// TIA Portal V16 export
// export: Created 2023-05-31T09:36:56.6738296Z, ExportSetting WithDefaults, DisplayName Totally Integrated Automation Portal, DisplayVersion V16 Update 3, DisplayName TIA Portal Version Control Interface, DisplayVersion V16 Update 2, DisplayName TIA Portal Openness, DisplayVersion V16 Update 3, DisplayName SINAMICS Startdrive Advanced, DisplayVersion V16, DisplayName SINAMICS Startdrive G130, G150, S120, S150, SINAMICS MV, S210, DisplayVersion V16, DisplayName SINAMICS Startdrive G110M, G120, G120C, G120D, G120P, DisplayVersion V16, DisplayName STEP 7 Professional, DisplayVersion V16 Update 3, DisplayName STEP 7 Safety, DisplayVersion V16, DisplayName WinCC Advanced, DisplayVersion V16 Update 3
FUNCTION "CIP LINEA 2" : Void   // FC54, LAD
{ S7_Optimized_Access := 'FALSE' }
VERSION : 0.1
// trabajo paralelo desde kjsdfgvjosod
// stored: AutoNumber false, IsIECCheckEnabled false, SetENOAutomatically false, UDAEnableTagReadback false
   VAR_TEMP   // added for the SCL form of the ladder/FBD networks
      _w1 : Bool;
      _s5time1 : S5Time;
   END_VAR
BEGIN

REGION Network 1: SOLO EN LIMPIEZA TANQUES
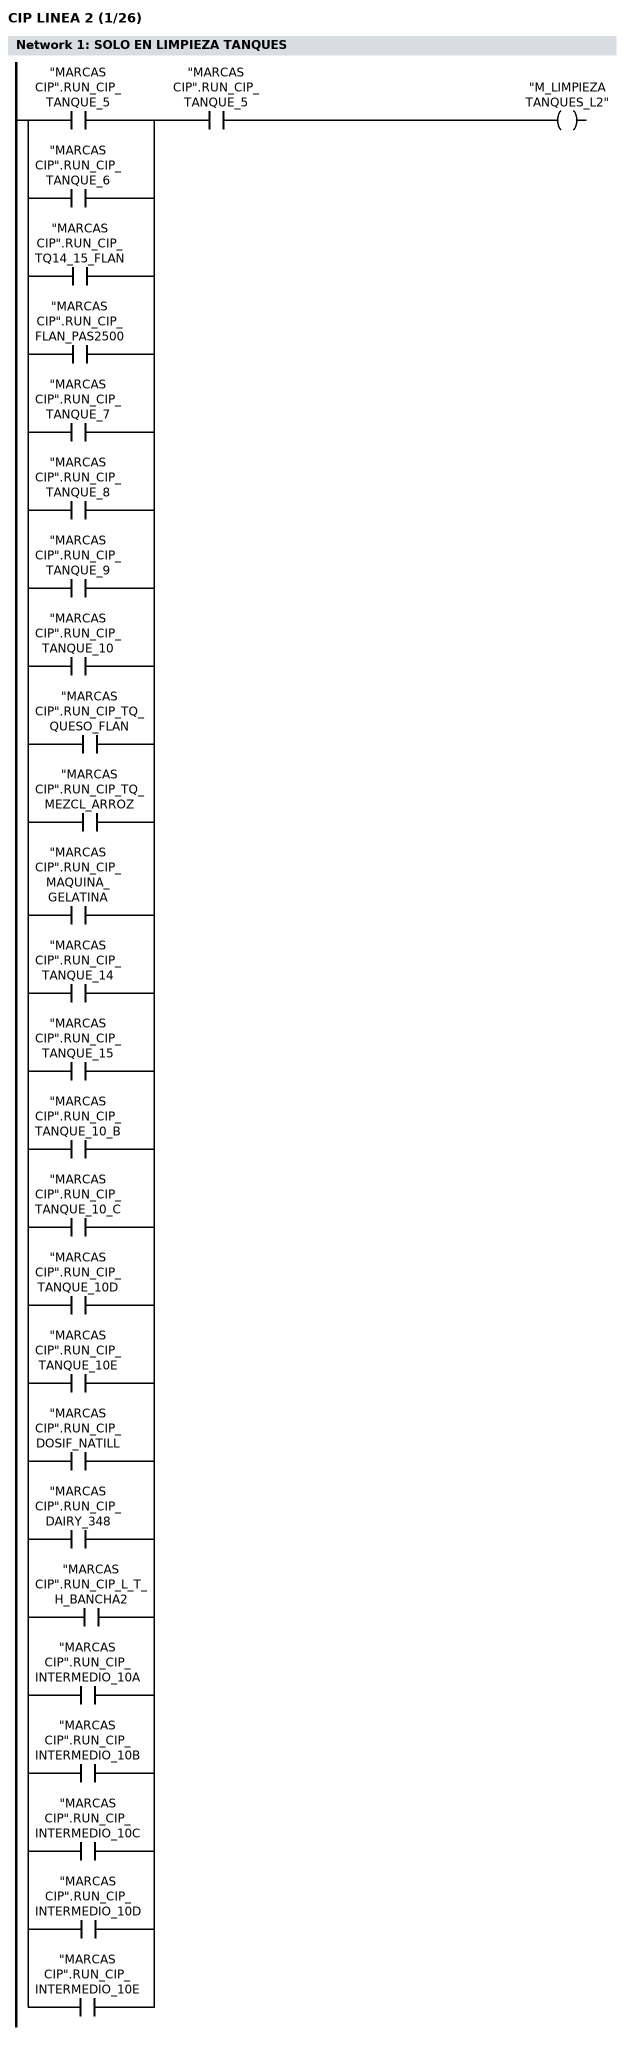
   RUNG wire#powerrail
      Contact( "MARCAS CIP".RUN_CIP_TANQUE_5 )
      wire#w1
      Contact( "MARCAS CIP".RUN_CIP_TANQUE_5 )
      Coil( "M_LIMPIEZA TANQUES_L2" )
   END_RUNG
   RUNG wire#powerrail
      Contact( "MARCAS CIP".RUN_CIP_TANQUE_6 )
   END_RUNG wire#w1
   RUNG wire#powerrail
      Contact( "MARCAS CIP".RUN_CIP_TQ14_15_FLAN )
   END_RUNG wire#w1
   RUNG wire#powerrail
      Contact( "MARCAS CIP".RUN_CIP_FLAN_PAS2500 )
   END_RUNG wire#w1
   RUNG wire#powerrail
      Contact( "MARCAS CIP".RUN_CIP_TANQUE_7 )
   END_RUNG wire#w1
   RUNG wire#powerrail
      Contact( "MARCAS CIP".RUN_CIP_TANQUE_8 )
   END_RUNG wire#w1
   RUNG wire#powerrail
      Contact( "MARCAS CIP".RUN_CIP_TANQUE_9 )
   END_RUNG wire#w1
   RUNG wire#powerrail
      Contact( "MARCAS CIP".RUN_CIP_TANQUE_10 )
   END_RUNG wire#w1
   RUNG wire#powerrail
      Contact( "MARCAS CIP".RUN_CIP_TQ_QUESO_FLAN )
   END_RUNG wire#w1
   RUNG wire#powerrail
      Contact( "MARCAS CIP".RUN_CIP_TQ_MEZCL_ARROZ )
   END_RUNG wire#w1
   RUNG wire#powerrail
      Contact( "MARCAS CIP".RUN_CIP_MAQUINA_GELATINA )
   END_RUNG wire#w1
   RUNG wire#powerrail
      Contact( "MARCAS CIP".RUN_CIP_TANQUE_14 )
   END_RUNG wire#w1
   RUNG wire#powerrail
      Contact( "MARCAS CIP".RUN_CIP_TANQUE_15 )
   END_RUNG wire#w1
   RUNG wire#powerrail
      Contact( "MARCAS CIP".RUN_CIP_TANQUE_10_B )
   END_RUNG wire#w1
   RUNG wire#powerrail
      Contact( "MARCAS CIP".RUN_CIP_TANQUE_10_C )
   END_RUNG wire#w1
   RUNG wire#powerrail
      Contact( "MARCAS CIP".RUN_CIP_TANQUE_10D )
   END_RUNG wire#w1
   RUNG wire#powerrail
      Contact( "MARCAS CIP".RUN_CIP_TANQUE_10E )
   END_RUNG wire#w1
   RUNG wire#powerrail
      Contact( "MARCAS CIP".RUN_CIP_DOSIF_NATILL )
   END_RUNG wire#w1
   RUNG wire#powerrail
      Contact( "MARCAS CIP".RUN_CIP_DAIRY_348 )
   END_RUNG wire#w1
   RUNG wire#powerrail
      Contact( "MARCAS CIP".RUN_CIP_L_T_H_BANCHA2 )
   END_RUNG wire#w1
   RUNG wire#powerrail
      Contact( "MARCAS CIP".RUN_CIP_INTERMEDIO_10A )
   END_RUNG wire#w1
   RUNG wire#powerrail
      Contact( "MARCAS CIP".RUN_CIP_INTERMEDIO_10B )
   END_RUNG wire#w1
   RUNG wire#powerrail
      Contact( "MARCAS CIP".RUN_CIP_INTERMEDIO_10C )
   END_RUNG wire#w1
   RUNG wire#powerrail
      Contact( "MARCAS CIP".RUN_CIP_INTERMEDIO_10D )
   END_RUNG wire#w1
   RUNG wire#powerrail
      Contact( "MARCAS CIP".RUN_CIP_INTERMEDIO_10E )
   END_RUNG wire#w1
   // the same network as SCL:
   "M_LIMPIEZA TANQUES_L2" := ("MARCAS CIP".RUN_CIP_TANQUE_5 OR "MARCAS CIP".RUN_CIP_TANQUE_6 OR "MARCAS CIP".RUN_CIP_TQ14_15_FLAN OR "MARCAS CIP".RUN_CIP_FLAN_PAS2500 OR "MARCAS CIP".RUN_CIP_TANQUE_7 OR "MARCAS CIP".RUN_CIP_TANQUE_8 OR "MARCAS CIP".RUN_CIP_TANQUE_9 OR "MARCAS CIP".RUN_CIP_TANQUE_10 OR "MARCAS CIP".RUN_CIP_TQ_QUESO_FLAN OR "MARCAS CIP".RUN_CIP_TQ_MEZCL_ARROZ OR "MARCAS CIP".RUN_CIP_MAQUINA_GELATINA OR "MARCAS CIP".RUN_CIP_TANQUE_14 OR "MARCAS CIP".RUN_CIP_TANQUE_15 OR "MARCAS CIP".RUN_CIP_TANQUE_10_B OR "MARCAS CIP".RUN_CIP_TANQUE_10_C OR "MARCAS CIP".RUN_CIP_TANQUE_10D OR "MARCAS CIP".RUN_CIP_TANQUE_10E OR "MARCAS CIP".RUN_CIP_DOSIF_NATILL OR "MARCAS CIP".RUN_CIP_DAIRY_348 OR "MARCAS CIP".RUN_CIP_L_T_H_BANCHA2 OR "MARCAS CIP".RUN_CIP_INTERMEDIO_10A OR "MARCAS CIP".RUN_CIP_INTERMEDIO_10B OR "MARCAS CIP".RUN_CIP_INTERMEDIO_10C OR "MARCAS CIP".RUN_CIP_INTERMEDIO_10D OR "MARCAS CIP".RUN_CIP_INTERMEDIO_10E) AND "MARCAS CIP".RUN_CIP_TANQUE_5;
END_REGION

REGION Network 2: PASO 1 PRIEMER ENJUAGUE AGUA RECUPERADA
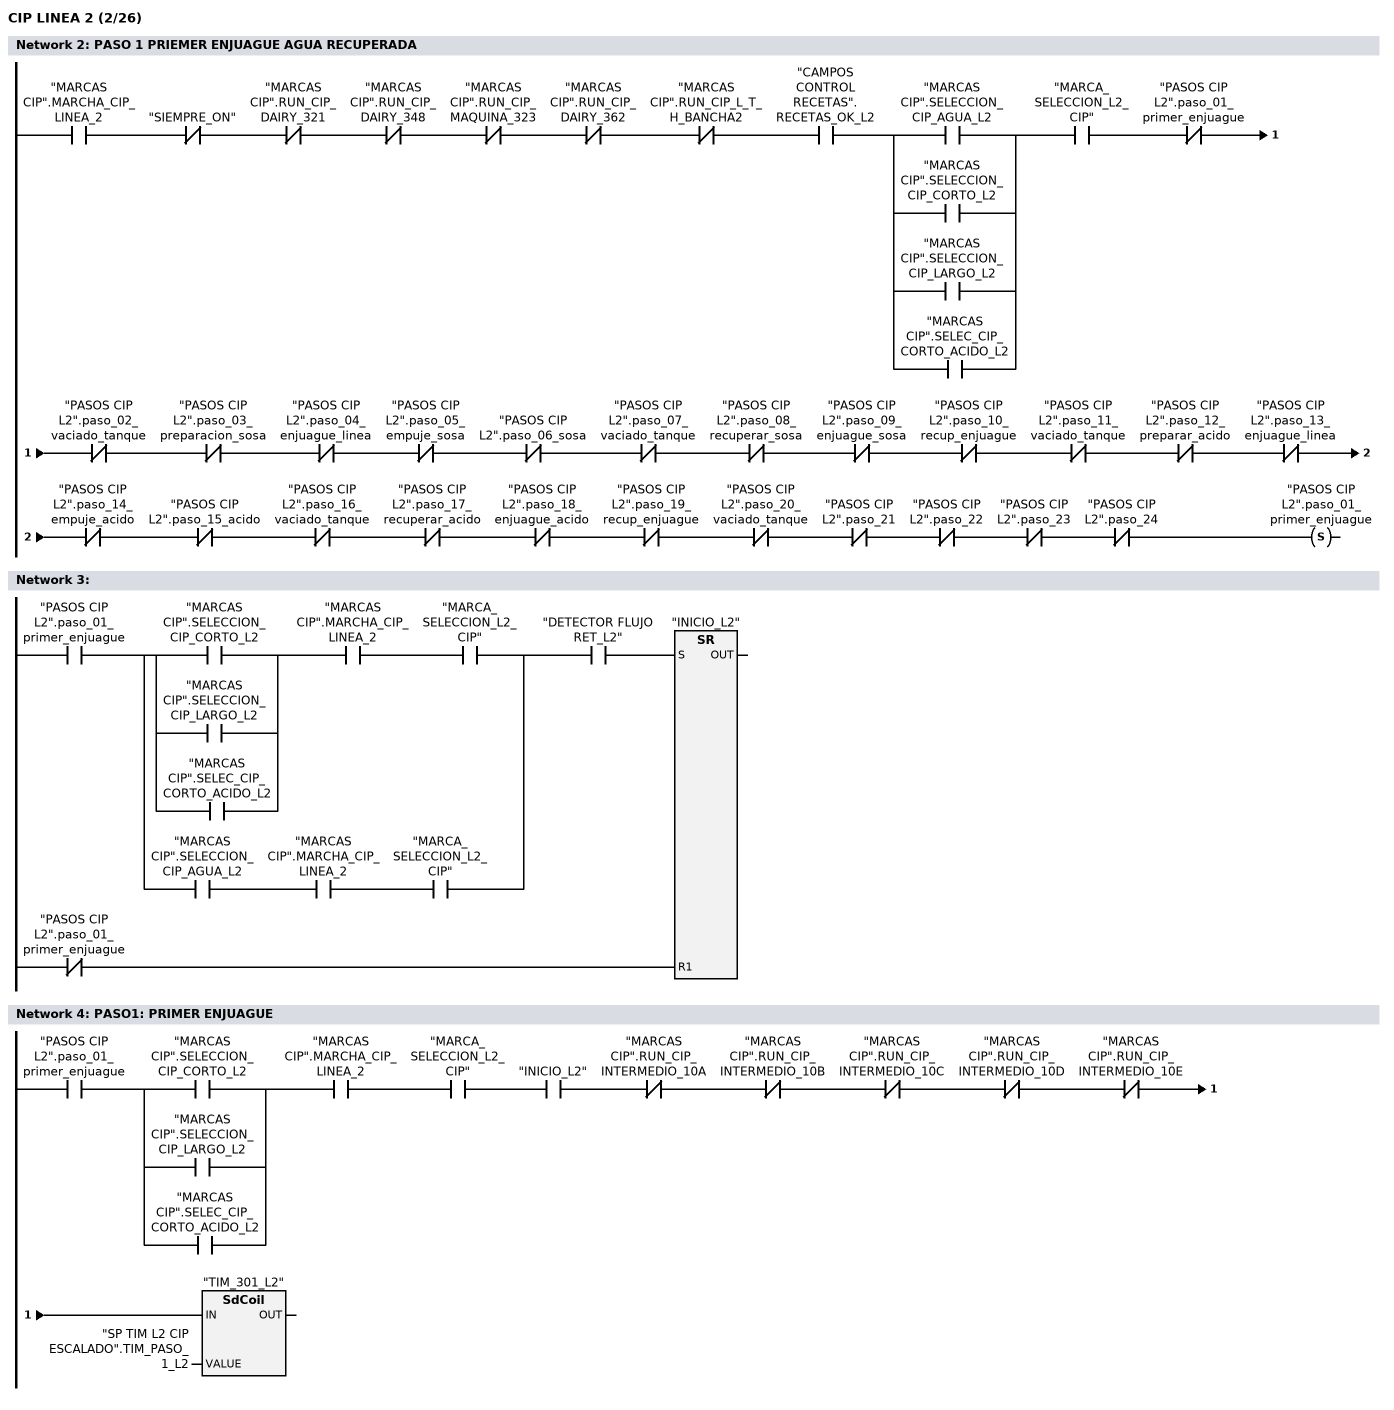
   RUNG wire#powerrail
      Contact( "MARCAS CIP".MARCHA_CIP_LINEA_2 )
      I_Contact( "SIEMPRE_ON" )
      I_Contact( "MARCAS CIP".RUN_CIP_DAIRY_321 )
      I_Contact( "MARCAS CIP".RUN_CIP_DAIRY_348 )
      I_Contact( "MARCAS CIP".RUN_CIP_MAQUINA_323 )
      I_Contact( "MARCAS CIP".RUN_CIP_DAIRY_362 )
      I_Contact( "MARCAS CIP".RUN_CIP_L_T_H_BANCHA2 )
      Contact( "CAMPOS CONTROL RECETAS".RECETAS_OK_L2 )
      wire#w1
      Contact( "MARCAS CIP".SELECCION_CIP_AGUA_L2 )
      wire#w2
      Contact( "MARCA_SELECCION_L2_CIP" )
      I_Contact( "PASOS CIP L2".paso_01_primer_enjuague )
      I_Contact( "PASOS CIP L2".paso_02_vaciado_tanque )
      I_Contact( "PASOS CIP L2".paso_03_preparacion_sosa )
      I_Contact( "PASOS CIP L2".paso_04_enjuague_linea )
      I_Contact( "PASOS CIP L2".paso_05_empuje_sosa )
      I_Contact( "PASOS CIP L2".paso_06_sosa )
      I_Contact( "PASOS CIP L2".paso_07_vaciado_tanque )
      I_Contact( "PASOS CIP L2".paso_08_recuperar_sosa )
      I_Contact( "PASOS CIP L2".paso_09_enjuague_sosa )
      I_Contact( "PASOS CIP L2".paso_10_recup_enjuague )
      I_Contact( "PASOS CIP L2".paso_11_vaciado_tanque )
      I_Contact( "PASOS CIP L2".paso_12_preparar_acido )
      I_Contact( "PASOS CIP L2".paso_13_enjuague_linea )
      I_Contact( "PASOS CIP L2".paso_14_empuje_acido )
      I_Contact( "PASOS CIP L2".paso_15_acido )
      I_Contact( "PASOS CIP L2".paso_16_vaciado_tanque )
      I_Contact( "PASOS CIP L2".paso_17_recuperar_acido )
      I_Contact( "PASOS CIP L2".paso_18_enjuague_acido )
      I_Contact( "PASOS CIP L2".paso_19_recup_enjuague )
      I_Contact( "PASOS CIP L2".paso_20_vaciado_tanque )
      I_Contact( "PASOS CIP L2".paso_21 )
      I_Contact( "PASOS CIP L2".paso_22 )
      I_Contact( "PASOS CIP L2".paso_23 )
      I_Contact( "PASOS CIP L2".paso_24 )
      S_Coil( "PASOS CIP L2".paso_01_primer_enjuague )
   END_RUNG
   RUNG wire#w1
      Contact( "MARCAS CIP".SELECCION_CIP_CORTO_L2 )
   END_RUNG wire#w2
   RUNG wire#w1
      Contact( "MARCAS CIP".SELECCION_CIP_LARGO_L2 )
   END_RUNG wire#w2
   RUNG wire#w1
      Contact( "MARCAS CIP".SELEC_CIP_CORTO_ACIDO_L2 )
   END_RUNG wire#w2
   // the same network as SCL:
   IF "MARCAS CIP".MARCHA_CIP_LINEA_2 AND NOT "SIEMPRE_ON" AND NOT "MARCAS CIP".RUN_CIP_DAIRY_321 AND NOT "MARCAS CIP".RUN_CIP_DAIRY_348 AND NOT "MARCAS CIP".RUN_CIP_MAQUINA_323 AND NOT "MARCAS CIP".RUN_CIP_DAIRY_362 AND NOT "MARCAS CIP".RUN_CIP_L_T_H_BANCHA2 AND "CAMPOS CONTROL RECETAS".RECETAS_OK_L2 AND ("MARCAS CIP".SELECCION_CIP_AGUA_L2 OR "MARCAS CIP".SELECCION_CIP_CORTO_L2 OR "MARCAS CIP".SELECCION_CIP_LARGO_L2 OR "MARCAS CIP".SELEC_CIP_CORTO_ACIDO_L2) AND "MARCA_SELECCION_L2_CIP" AND NOT "PASOS CIP L2".paso_01_primer_enjuague AND NOT "PASOS CIP L2".paso_02_vaciado_tanque AND NOT "PASOS CIP L2".paso_03_preparacion_sosa AND NOT "PASOS CIP L2".paso_04_enjuague_linea AND NOT "PASOS CIP L2".paso_05_empuje_sosa AND NOT "PASOS CIP L2".paso_06_sosa AND NOT "PASOS CIP L2".paso_07_vaciado_tanque AND NOT "PASOS CIP L2".paso_08_recuperar_sosa AND NOT "PASOS CIP L2".paso_09_enjuague_sosa AND NOT "PASOS CIP L2".paso_10_recup_enjuague AND NOT "PASOS CIP L2".paso_11_vaciado_tanque AND NOT "PASOS CIP L2".paso_12_preparar_acido AND NOT "PASOS CIP L2".paso_13_enjuague_linea AND NOT "PASOS CIP L2".paso_14_empuje_acido AND NOT "PASOS CIP L2".paso_15_acido AND NOT "PASOS CIP L2".paso_16_vaciado_tanque AND NOT "PASOS CIP L2".paso_17_recuperar_acido AND NOT "PASOS CIP L2".paso_18_enjuague_acido AND NOT "PASOS CIP L2".paso_19_recup_enjuague AND NOT "PASOS CIP L2".paso_20_vaciado_tanque AND NOT "PASOS CIP L2".paso_21 AND NOT "PASOS CIP L2".paso_22 AND NOT "PASOS CIP L2".paso_23 AND NOT "PASOS CIP L2".paso_24 THEN
       "PASOS CIP L2".paso_01_primer_enjuague := TRUE;
   END_IF;
END_REGION

REGION Network 3
   RUNG wire#powerrail
      Contact( "PASOS CIP L2".paso_01_primer_enjuague )
      wire#w1
      Contact( "MARCAS CIP".SELECCION_CIP_CORTO_L2 )
      wire#w2
      Contact( "MARCAS CIP".MARCHA_CIP_LINEA_2 )
      Contact( "MARCA_SELECCION_L2_CIP" )
      wire#w3
      Contact( "DETECTOR FLUJO RET_L2" )
      S_SR(operand := "INICIO_L2", r1 := wire#w4)
   END_RUNG
   RUNG wire#w1
      Contact( "MARCAS CIP".SELECCION_CIP_LARGO_L2 )
   END_RUNG wire#w2
   RUNG wire#w1
      Contact( "MARCAS CIP".SELEC_CIP_CORTO_ACIDO_L2 )
   END_RUNG wire#w2
   RUNG wire#w1
      Contact( "MARCAS CIP".SELECCION_CIP_AGUA_L2 )
      Contact( "MARCAS CIP".MARCHA_CIP_LINEA_2 )
      Contact( "MARCA_SELECCION_L2_CIP" )
   END_RUNG wire#w3
   RUNG wire#powerrail
      I_Contact( "PASOS CIP L2".paso_01_primer_enjuague )
   END_RUNG wire#w4
   // the same network as SCL:
   IF "PASOS CIP L2".paso_01_primer_enjuague AND ((("MARCAS CIP".SELECCION_CIP_CORTO_L2 OR "MARCAS CIP".SELECCION_CIP_LARGO_L2 OR "MARCAS CIP".SELEC_CIP_CORTO_ACIDO_L2) AND "MARCAS CIP".MARCHA_CIP_LINEA_2 AND "MARCA_SELECCION_L2_CIP") OR ("MARCAS CIP".SELECCION_CIP_AGUA_L2 AND "MARCAS CIP".MARCHA_CIP_LINEA_2 AND "MARCA_SELECCION_L2_CIP")) AND "DETECTOR FLUJO RET_L2" THEN
       "INICIO_L2" := TRUE;   // SR flip-flop
   END_IF;
   IF NOT "PASOS CIP L2".paso_01_primer_enjuague THEN "INICIO_L2" := FALSE; END_IF;
END_REGION

REGION Network 4: PASO1: PRIMER ENJUAGUE
   // no SCL statement known for SdCoil: written as a call
   SdCoil(value := "SP TIM L2 CIP ESCALADO".TIM_PASO_1_L2,
          operand := "TIM_301_L2",
          in := "PASOS CIP L2".paso_01_primer_enjuague AND ("MARCAS CIP".SELECCION_CIP_CORTO_L2 OR "MARCAS CIP".SELECCION_CIP_LARGO_L2 OR "MARCAS CIP".SELEC_CIP_CORTO_ACIDO_L2) AND "MARCAS CIP".MARCHA_CIP_LINEA_2 AND "MARCA_SELECCION_L2_CIP" AND "INICIO_L2" AND NOT "MARCAS CIP".RUN_CIP_INTERMEDIO_10A AND NOT "MARCAS CIP".RUN_CIP_INTERMEDIO_10B AND NOT "MARCAS CIP".RUN_CIP_INTERMEDIO_10C AND NOT "MARCAS CIP".RUN_CIP_INTERMEDIO_10D AND NOT "MARCAS CIP".RUN_CIP_INTERMEDIO_10E);
END_REGION

REGION Network 5: PASO 2: VACIADO TANQUE (SOLO BOMBA RETORNO CIP)
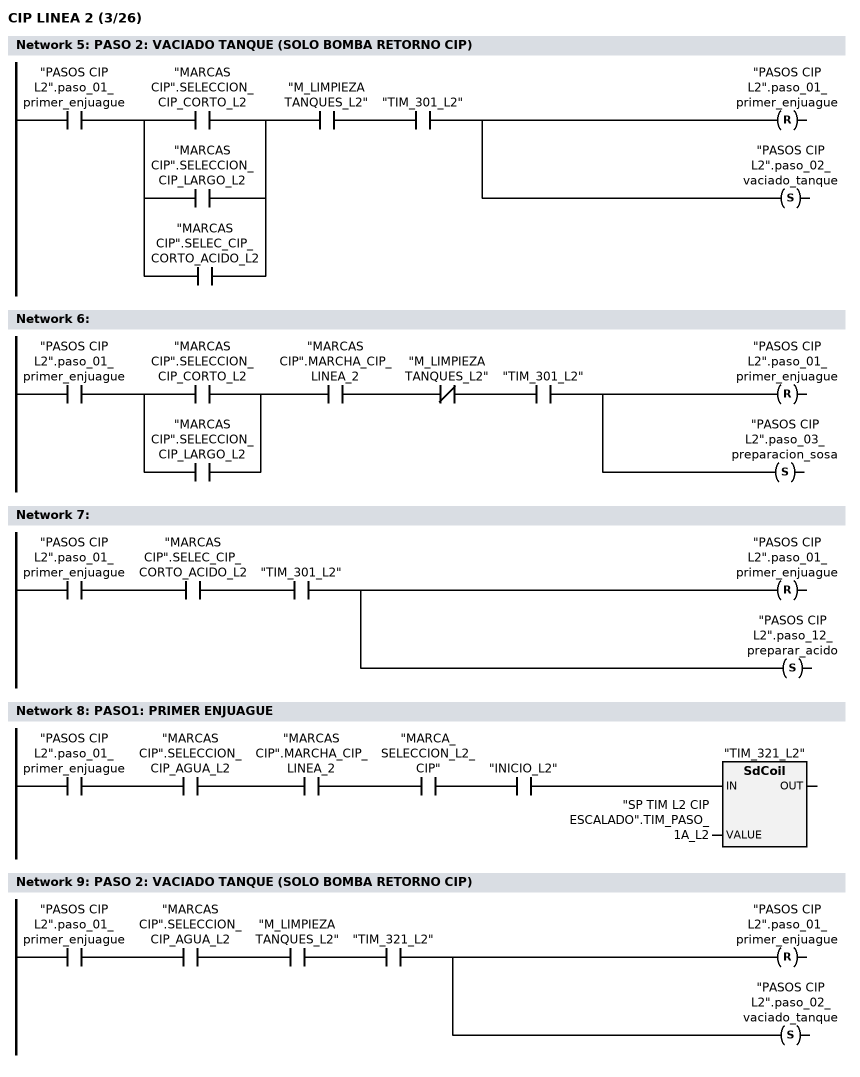
   RUNG wire#powerrail
      Contact( "PASOS CIP L2".paso_01_primer_enjuague )
      wire#w1
      Contact( "MARCAS CIP".SELECCION_CIP_CORTO_L2 )
      wire#w2
      Contact( "M_LIMPIEZA TANQUES_L2" )
      Contact( "TIM_301_L2" )
      wire#w3
      R_Coil( "PASOS CIP L2".paso_01_primer_enjuague )
   END_RUNG
   RUNG wire#w1
      Contact( "MARCAS CIP".SELECCION_CIP_LARGO_L2 )
   END_RUNG wire#w2
   RUNG wire#w1
      Contact( "MARCAS CIP".SELEC_CIP_CORTO_ACIDO_L2 )
   END_RUNG wire#w2
   RUNG wire#w3
      S_Coil( "PASOS CIP L2".paso_02_vaciado_tanque )
   END_RUNG
   // the same network as SCL:
   #_w1 := "PASOS CIP L2".paso_01_primer_enjuague AND ("MARCAS CIP".SELECCION_CIP_CORTO_L2 OR "MARCAS CIP".SELECCION_CIP_LARGO_L2 OR "MARCAS CIP".SELEC_CIP_CORTO_ACIDO_L2) AND "M_LIMPIEZA TANQUES_L2" AND "TIM_301_L2";
   IF #_w1 THEN
       "PASOS CIP L2".paso_01_primer_enjuague := FALSE;
       "PASOS CIP L2".paso_02_vaciado_tanque := TRUE;
   END_IF;
END_REGION

REGION Network 6
   RUNG wire#powerrail
      Contact( "PASOS CIP L2".paso_01_primer_enjuague )
      wire#w1
      Contact( "MARCAS CIP".SELECCION_CIP_CORTO_L2 )
      wire#w2
      Contact( "MARCAS CIP".MARCHA_CIP_LINEA_2 )
      I_Contact( "M_LIMPIEZA TANQUES_L2" )
      Contact( "TIM_301_L2" )
      wire#w3
      R_Coil( "PASOS CIP L2".paso_01_primer_enjuague )
   END_RUNG
   RUNG wire#w1
      Contact( "MARCAS CIP".SELECCION_CIP_LARGO_L2 )
   END_RUNG wire#w2
   RUNG wire#w3
      S_Coil( "PASOS CIP L2".paso_03_preparacion_sosa )
   END_RUNG
   // the same network as SCL:
   #_w1 := "PASOS CIP L2".paso_01_primer_enjuague AND ("MARCAS CIP".SELECCION_CIP_CORTO_L2 OR "MARCAS CIP".SELECCION_CIP_LARGO_L2) AND "MARCAS CIP".MARCHA_CIP_LINEA_2 AND NOT "M_LIMPIEZA TANQUES_L2" AND "TIM_301_L2";
   IF #_w1 THEN
       "PASOS CIP L2".paso_01_primer_enjuague := FALSE;
       "PASOS CIP L2".paso_03_preparacion_sosa := TRUE;
   END_IF;
END_REGION

REGION Network 7
   RUNG wire#powerrail
      Contact( "PASOS CIP L2".paso_01_primer_enjuague )
      Contact( "MARCAS CIP".SELEC_CIP_CORTO_ACIDO_L2 )
      Contact( "TIM_301_L2" )
      wire#w1
      R_Coil( "PASOS CIP L2".paso_01_primer_enjuague )
   END_RUNG
   RUNG wire#w1
      S_Coil( "PASOS CIP L2".paso_12_preparar_acido )
   END_RUNG
   // the same network as SCL:
   #_w1 := "PASOS CIP L2".paso_01_primer_enjuague AND "MARCAS CIP".SELEC_CIP_CORTO_ACIDO_L2 AND "TIM_301_L2";
   IF #_w1 THEN
       "PASOS CIP L2".paso_01_primer_enjuague := FALSE;
       "PASOS CIP L2".paso_12_preparar_acido := TRUE;
   END_IF;
END_REGION

REGION Network 8: PASO1: PRIMER ENJUAGUE
   // no SCL statement known for SdCoil: written as a call
   SdCoil(value := "SP TIM L2 CIP ESCALADO".TIM_PASO_1A_L2,
          operand := "TIM_321_L2",
          in := "PASOS CIP L2".paso_01_primer_enjuague AND "MARCAS CIP".SELECCION_CIP_AGUA_L2 AND "MARCAS CIP".MARCHA_CIP_LINEA_2 AND "MARCA_SELECCION_L2_CIP" AND "INICIO_L2");
END_REGION

REGION Network 9: PASO 2: VACIADO TANQUE (SOLO BOMBA RETORNO CIP)
   RUNG wire#powerrail
      Contact( "PASOS CIP L2".paso_01_primer_enjuague )
      Contact( "MARCAS CIP".SELECCION_CIP_AGUA_L2 )
      Contact( "M_LIMPIEZA TANQUES_L2" )
      Contact( "TIM_321_L2" )
      wire#w1
      R_Coil( "PASOS CIP L2".paso_01_primer_enjuague )
   END_RUNG
   RUNG wire#w1
      S_Coil( "PASOS CIP L2".paso_02_vaciado_tanque )
   END_RUNG
   // the same network as SCL:
   #_w1 := "PASOS CIP L2".paso_01_primer_enjuague AND "MARCAS CIP".SELECCION_CIP_AGUA_L2 AND "M_LIMPIEZA TANQUES_L2" AND "TIM_321_L2";
   IF #_w1 THEN
       "PASOS CIP L2".paso_01_primer_enjuague := FALSE;
       "PASOS CIP L2".paso_02_vaciado_tanque := TRUE;
   END_IF;
END_REGION

REGION Network 10
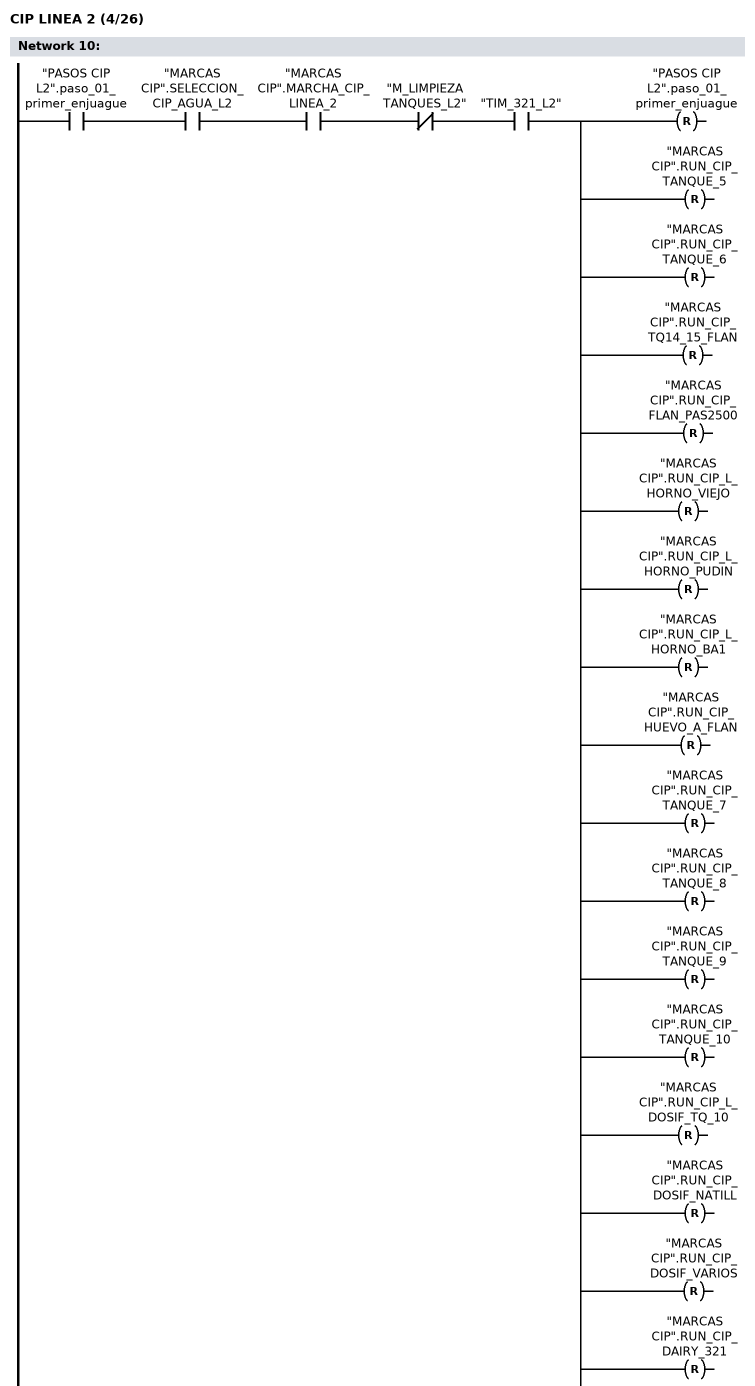
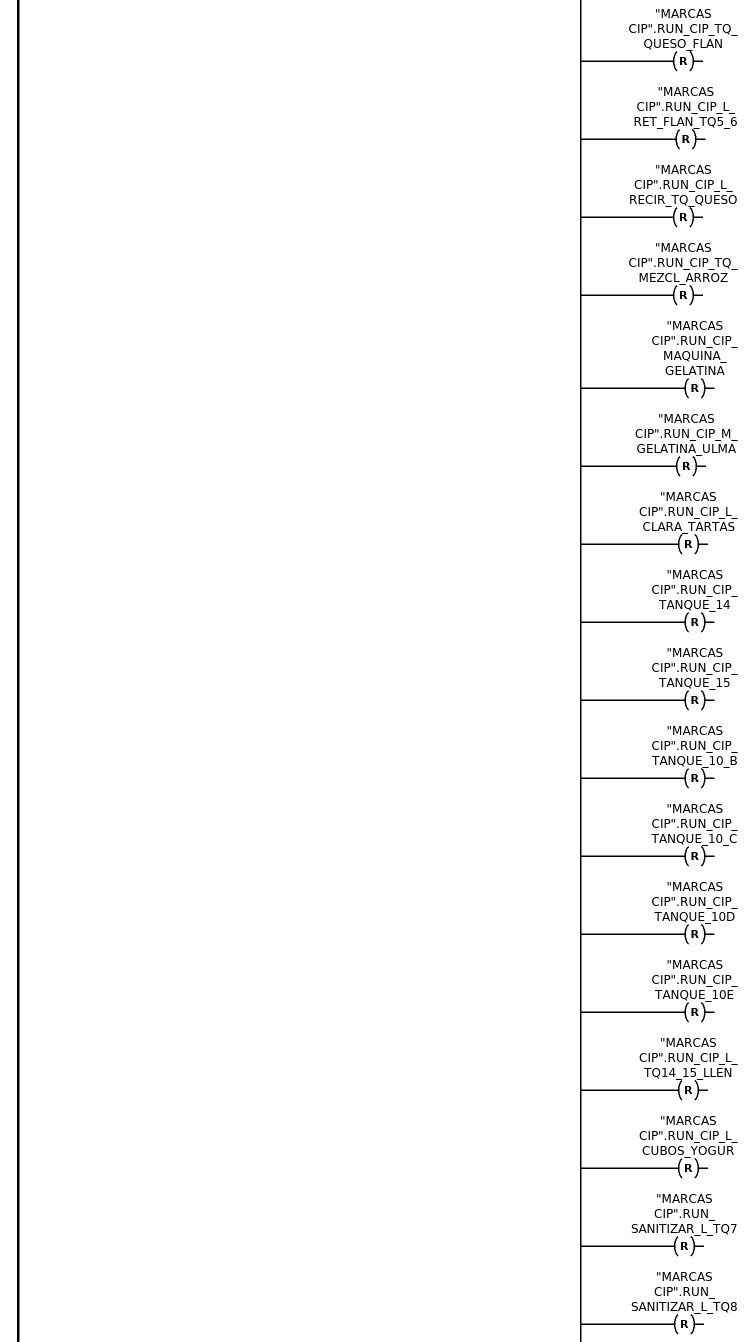
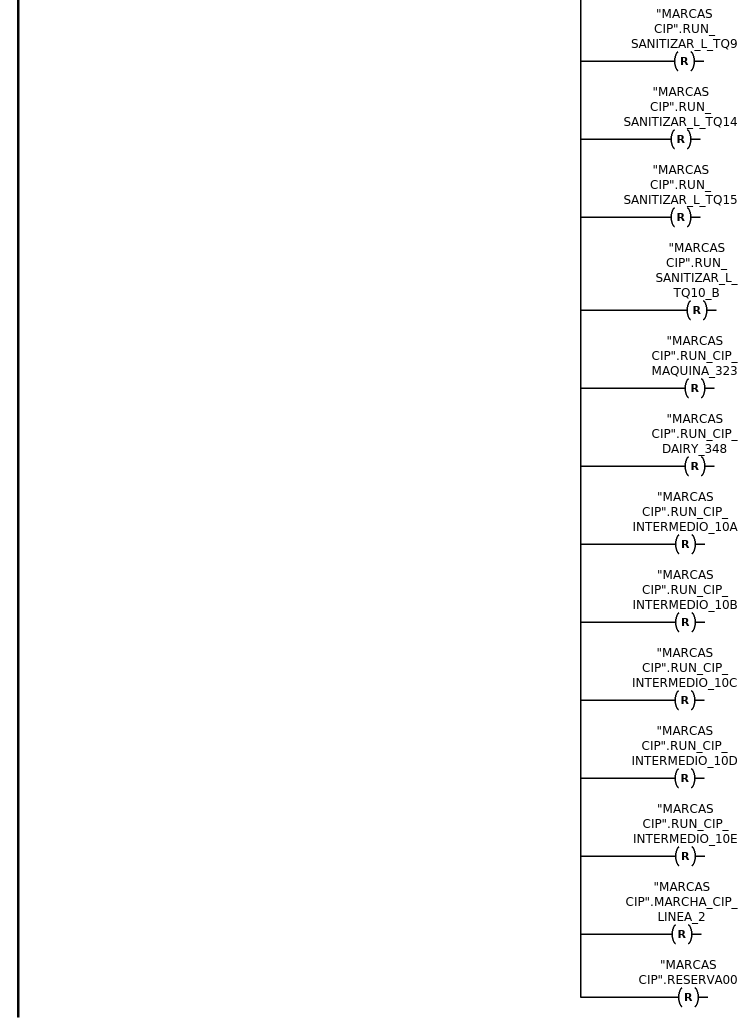
   RUNG wire#powerrail
      Contact( "PASOS CIP L2".paso_01_primer_enjuague )
      Contact( "MARCAS CIP".SELECCION_CIP_AGUA_L2 )
      Contact( "MARCAS CIP".MARCHA_CIP_LINEA_2 )
      I_Contact( "M_LIMPIEZA TANQUES_L2" )
      Contact( "TIM_321_L2" )
      wire#w1
      R_Coil( "PASOS CIP L2".paso_01_primer_enjuague )
   END_RUNG
   RUNG wire#w1
      R_Coil( "MARCAS CIP".RUN_CIP_TANQUE_5 )
   END_RUNG
   RUNG wire#w1
      R_Coil( "MARCAS CIP".RUN_CIP_TANQUE_6 )
   END_RUNG
   RUNG wire#w1
      R_Coil( "MARCAS CIP".RUN_CIP_TQ14_15_FLAN )
   END_RUNG
   RUNG wire#w1
      R_Coil( "MARCAS CIP".RUN_CIP_FLAN_PAS2500 )
   END_RUNG
   RUNG wire#w1
      R_Coil( "MARCAS CIP".RUN_CIP_L_HORNO_VIEJO )
   END_RUNG
   RUNG wire#w1
      R_Coil( "MARCAS CIP".RUN_CIP_L_HORNO_PUDIN )
   END_RUNG
   RUNG wire#w1
      R_Coil( "MARCAS CIP".RUN_CIP_L_HORNO_BA1 )
   END_RUNG
   RUNG wire#w1
      R_Coil( "MARCAS CIP".RUN_CIP_HUEVO_A_FLAN )
   END_RUNG
   RUNG wire#w1
      R_Coil( "MARCAS CIP".RUN_CIP_TANQUE_7 )
   END_RUNG
   RUNG wire#w1
      R_Coil( "MARCAS CIP".RUN_CIP_TANQUE_8 )
   END_RUNG
   RUNG wire#w1
      R_Coil( "MARCAS CIP".RUN_CIP_TANQUE_9 )
   END_RUNG
   RUNG wire#w1
      R_Coil( "MARCAS CIP".RUN_CIP_TANQUE_10 )
   END_RUNG
   RUNG wire#w1
      R_Coil( "MARCAS CIP".RUN_CIP_L_DOSIF_TQ_10 )
   END_RUNG
   RUNG wire#w1
      R_Coil( "MARCAS CIP".RUN_CIP_DOSIF_NATILL )
   END_RUNG
   RUNG wire#w1
      R_Coil( "MARCAS CIP".RUN_CIP_DOSIF_VARIOS )
   END_RUNG
   RUNG wire#w1
      R_Coil( "MARCAS CIP".RUN_CIP_DAIRY_321 )
   END_RUNG
   RUNG wire#w1
      R_Coil( "MARCAS CIP".RUN_CIP_TQ_QUESO_FLAN )
   END_RUNG
   RUNG wire#w1
      R_Coil( "MARCAS CIP".RUN_CIP_L_RET_FLAN_TQ5_6 )
   END_RUNG
   RUNG wire#w1
      R_Coil( "MARCAS CIP".RUN_CIP_L_RECIR_TQ_QUESO )
   END_RUNG
   RUNG wire#w1
      R_Coil( "MARCAS CIP".RUN_CIP_TQ_MEZCL_ARROZ )
   END_RUNG
   RUNG wire#w1
      R_Coil( "MARCAS CIP".RUN_CIP_MAQUINA_GELATINA )
   END_RUNG
   RUNG wire#w1
      R_Coil( "MARCAS CIP".RUN_CIP_M_GELATINA_ULMA )
   END_RUNG
   RUNG wire#w1
      R_Coil( "MARCAS CIP".RUN_CIP_L_CLARA_TARTAS )
   END_RUNG
   RUNG wire#w1
      R_Coil( "MARCAS CIP".RUN_CIP_TANQUE_14 )
   END_RUNG
   RUNG wire#w1
      R_Coil( "MARCAS CIP".RUN_CIP_TANQUE_15 )
   END_RUNG
   RUNG wire#w1
      R_Coil( "MARCAS CIP".RUN_CIP_TANQUE_10_B )
   END_RUNG
   RUNG wire#w1
      R_Coil( "MARCAS CIP".RUN_CIP_TANQUE_10_C )
   END_RUNG
   RUNG wire#w1
      R_Coil( "MARCAS CIP".RUN_CIP_TANQUE_10D )
   END_RUNG
   RUNG wire#w1
      R_Coil( "MARCAS CIP".RUN_CIP_TANQUE_10E )
   END_RUNG
   RUNG wire#w1
      R_Coil( "MARCAS CIP".RUN_CIP_L_TQ14_15_LLEN )
   END_RUNG
   RUNG wire#w1
      R_Coil( "MARCAS CIP".RUN_CIP_L_CUBOS_YOGUR )
   END_RUNG
   RUNG wire#w1
      R_Coil( "MARCAS CIP".RUN_SANITIZAR_L_TQ7 )
   END_RUNG
   RUNG wire#w1
      R_Coil( "MARCAS CIP".RUN_SANITIZAR_L_TQ8 )
   END_RUNG
   RUNG wire#w1
      R_Coil( "MARCAS CIP".RUN_SANITIZAR_L_TQ9 )
   END_RUNG
   RUNG wire#w1
      R_Coil( "MARCAS CIP".RUN_SANITIZAR_L_TQ14 )
   END_RUNG
   RUNG wire#w1
      R_Coil( "MARCAS CIP".RUN_SANITIZAR_L_TQ15 )
   END_RUNG
   RUNG wire#w1
      R_Coil( "MARCAS CIP".RUN_SANITIZAR_L_TQ10_B )
   END_RUNG
   RUNG wire#w1
      R_Coil( "MARCAS CIP".RUN_CIP_MAQUINA_323 )
   END_RUNG
   RUNG wire#w1
      R_Coil( "MARCAS CIP".RUN_CIP_DAIRY_348 )
   END_RUNG
   RUNG wire#w1
      R_Coil( "MARCAS CIP".RUN_CIP_INTERMEDIO_10A )
   END_RUNG
   RUNG wire#w1
      R_Coil( "MARCAS CIP".RUN_CIP_INTERMEDIO_10B )
   END_RUNG
   RUNG wire#w1
      R_Coil( "MARCAS CIP".RUN_CIP_INTERMEDIO_10C )
   END_RUNG
   RUNG wire#w1
      R_Coil( "MARCAS CIP".RUN_CIP_INTERMEDIO_10D )
   END_RUNG
   RUNG wire#w1
      R_Coil( "MARCAS CIP".RUN_CIP_INTERMEDIO_10E )
   END_RUNG
   RUNG wire#w1
      R_Coil( "MARCAS CIP".MARCHA_CIP_LINEA_2 )
   END_RUNG
   RUNG wire#w1
      R_Coil( "MARCAS CIP".RESERVA00 )
   END_RUNG
   // the same network as SCL:
   #_w1 := "PASOS CIP L2".paso_01_primer_enjuague AND "MARCAS CIP".SELECCION_CIP_AGUA_L2 AND "MARCAS CIP".MARCHA_CIP_LINEA_2 AND NOT "M_LIMPIEZA TANQUES_L2" AND "TIM_321_L2";
   IF #_w1 THEN
       "PASOS CIP L2".paso_01_primer_enjuague := FALSE;
       "MARCAS CIP".RUN_CIP_TANQUE_5 := FALSE;
       "MARCAS CIP".RUN_CIP_TANQUE_6 := FALSE;
       "MARCAS CIP".RUN_CIP_TQ14_15_FLAN := FALSE;
       "MARCAS CIP".RUN_CIP_FLAN_PAS2500 := FALSE;
       "MARCAS CIP".RUN_CIP_L_HORNO_VIEJO := FALSE;
       "MARCAS CIP".RUN_CIP_L_HORNO_PUDIN := FALSE;
       "MARCAS CIP".RUN_CIP_L_HORNO_BA1 := FALSE;
       "MARCAS CIP".RUN_CIP_HUEVO_A_FLAN := FALSE;
       "MARCAS CIP".RUN_CIP_TANQUE_7 := FALSE;
       "MARCAS CIP".RUN_CIP_TANQUE_8 := FALSE;
       "MARCAS CIP".RUN_CIP_TANQUE_9 := FALSE;
       "MARCAS CIP".RUN_CIP_TANQUE_10 := FALSE;
       "MARCAS CIP".RUN_CIP_L_DOSIF_TQ_10 := FALSE;
       "MARCAS CIP".RUN_CIP_DOSIF_NATILL := FALSE;
       "MARCAS CIP".RUN_CIP_DOSIF_VARIOS := FALSE;
       "MARCAS CIP".RUN_CIP_DAIRY_321 := FALSE;
       "MARCAS CIP".RUN_CIP_TQ_QUESO_FLAN := FALSE;
       "MARCAS CIP".RUN_CIP_L_RET_FLAN_TQ5_6 := FALSE;
       "MARCAS CIP".RUN_CIP_L_RECIR_TQ_QUESO := FALSE;
       "MARCAS CIP".RUN_CIP_TQ_MEZCL_ARROZ := FALSE;
       "MARCAS CIP".RUN_CIP_MAQUINA_GELATINA := FALSE;
       "MARCAS CIP".RUN_CIP_M_GELATINA_ULMA := FALSE;
       "MARCAS CIP".RUN_CIP_L_CLARA_TARTAS := FALSE;
       "MARCAS CIP".RUN_CIP_TANQUE_14 := FALSE;
       "MARCAS CIP".RUN_CIP_TANQUE_15 := FALSE;
       "MARCAS CIP".RUN_CIP_TANQUE_10_B := FALSE;
       "MARCAS CIP".RUN_CIP_TANQUE_10_C := FALSE;
       "MARCAS CIP".RUN_CIP_TANQUE_10D := FALSE;
       "MARCAS CIP".RUN_CIP_TANQUE_10E := FALSE;
       "MARCAS CIP".RUN_CIP_L_TQ14_15_LLEN := FALSE;
       "MARCAS CIP".RUN_CIP_L_CUBOS_YOGUR := FALSE;
       "MARCAS CIP".RUN_SANITIZAR_L_TQ7 := FALSE;
       "MARCAS CIP".RUN_SANITIZAR_L_TQ8 := FALSE;
       "MARCAS CIP".RUN_SANITIZAR_L_TQ9 := FALSE;
       "MARCAS CIP".RUN_SANITIZAR_L_TQ14 := FALSE;
       "MARCAS CIP".RUN_SANITIZAR_L_TQ15 := FALSE;
       "MARCAS CIP".RUN_SANITIZAR_L_TQ10_B := FALSE;
       "MARCAS CIP".RUN_CIP_MAQUINA_323 := FALSE;
       "MARCAS CIP".RUN_CIP_DAIRY_348 := FALSE;
       "MARCAS CIP".RUN_CIP_INTERMEDIO_10A := FALSE;
       "MARCAS CIP".RUN_CIP_INTERMEDIO_10B := FALSE;
       "MARCAS CIP".RUN_CIP_INTERMEDIO_10C := FALSE;
       "MARCAS CIP".RUN_CIP_INTERMEDIO_10D := FALSE;
       "MARCAS CIP".RUN_CIP_INTERMEDIO_10E := FALSE;
       "MARCAS CIP".MARCHA_CIP_LINEA_2 := FALSE;
       "MARCAS CIP".RESERVA00 := FALSE;
   END_IF;
END_REGION

REGION Network 11
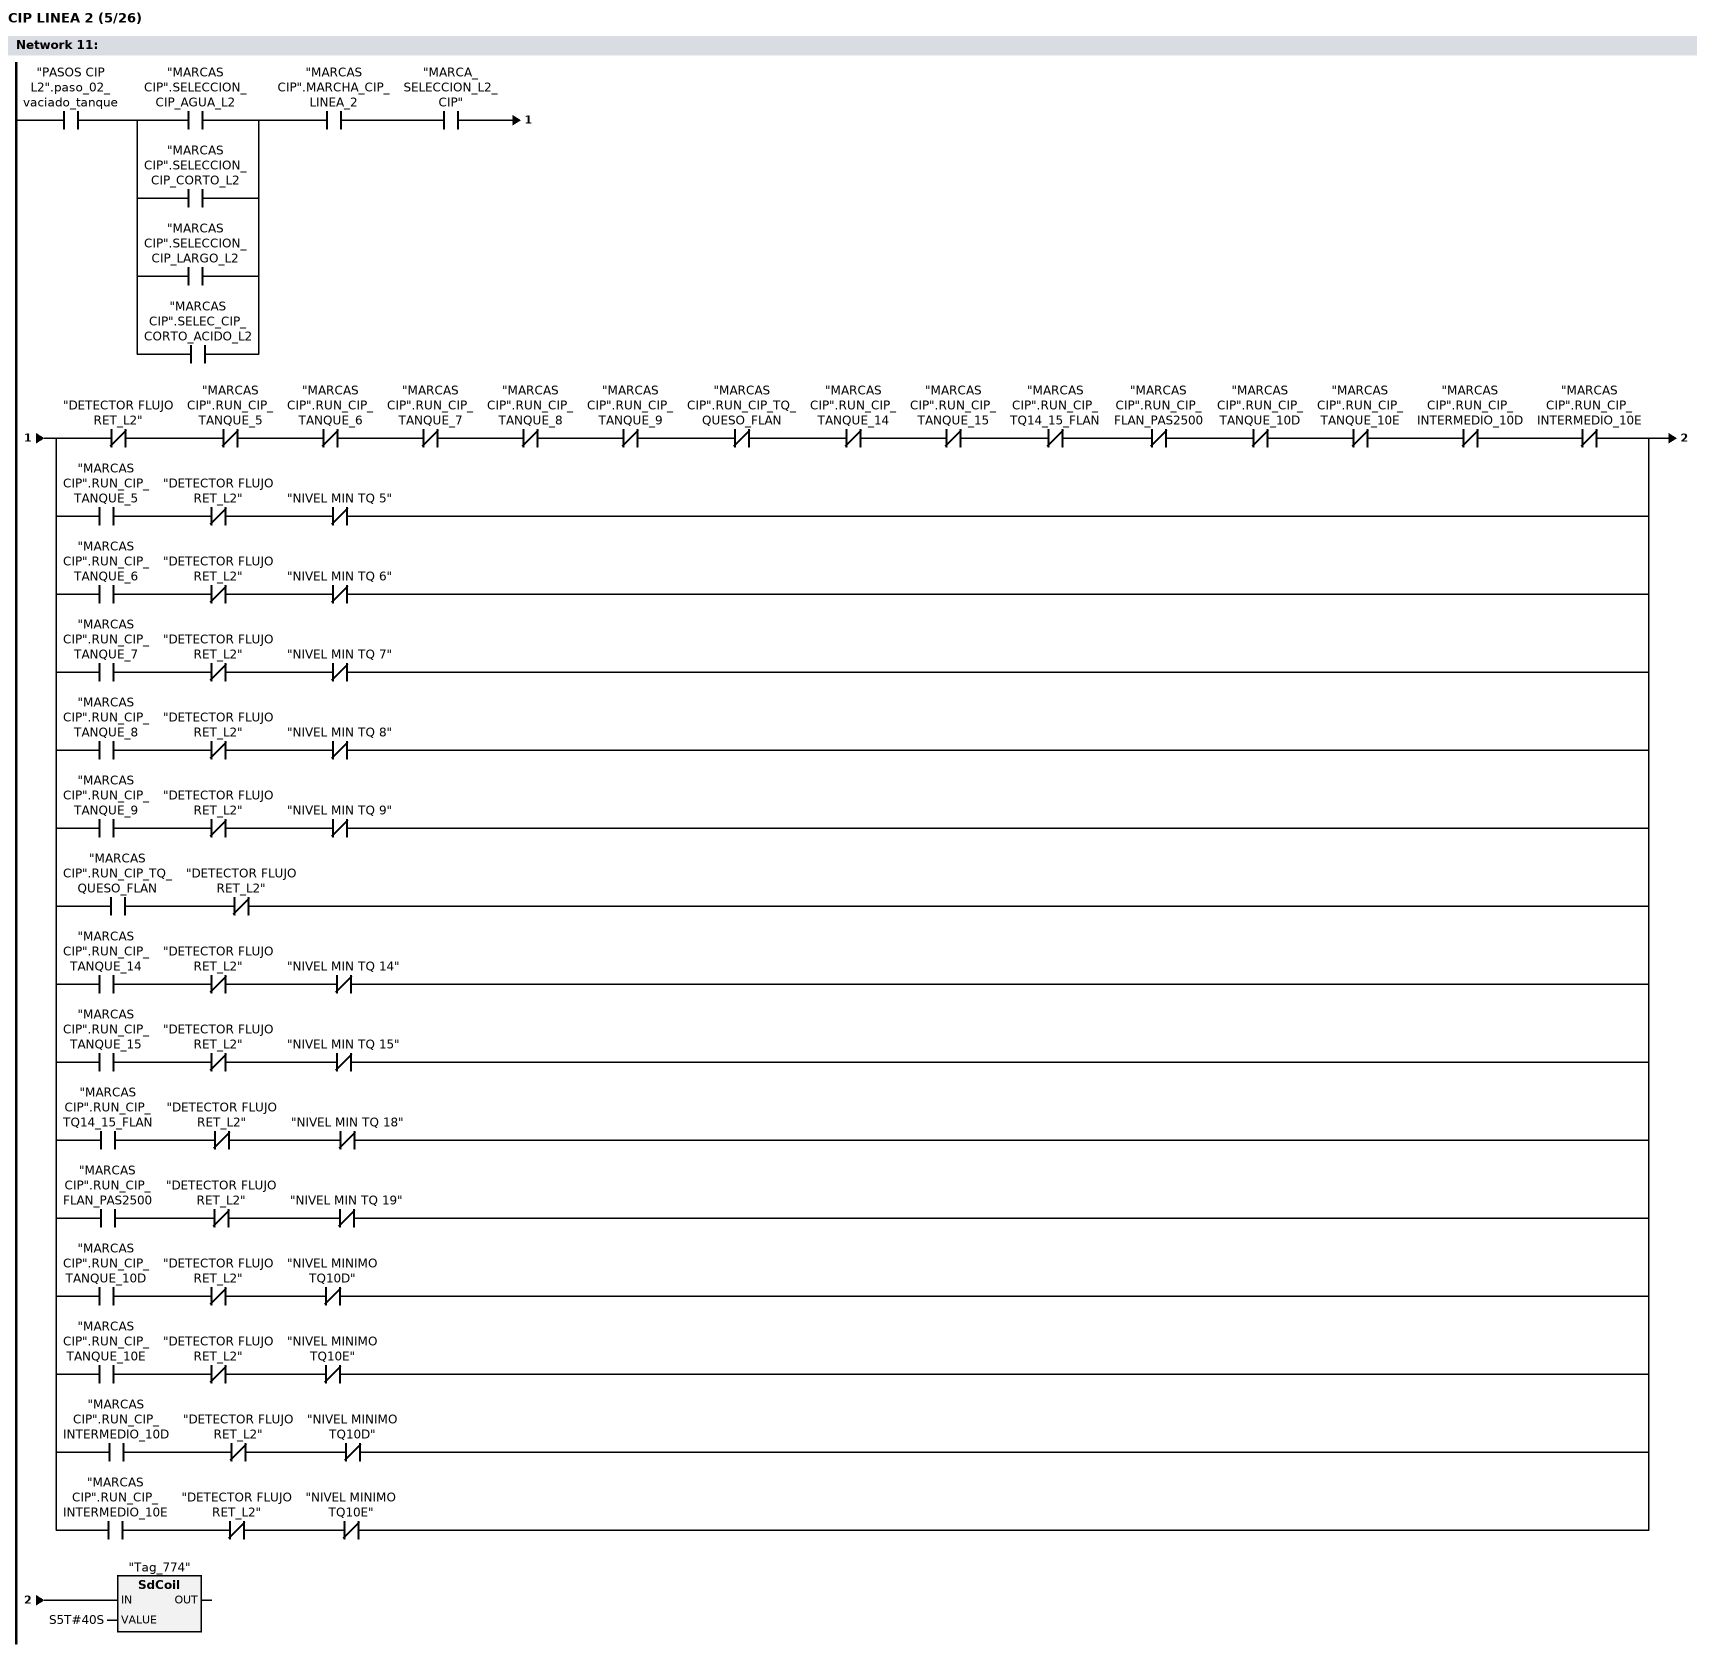
   // no SCL statement known for SdCoil: written as a call
   SdCoil(value := S5T#40S,
          in := "PASOS CIP L2".paso_02_vaciado_tanque AND ("MARCAS CIP".SELECCION_CIP_AGUA_L2 OR "MARCAS CIP".SELECCION_CIP_CORTO_L2 OR "MARCAS CIP".SELECCION_CIP_LARGO_L2 OR "MARCAS CIP".SELEC_CIP_CORTO_ACIDO_L2) AND "MARCAS CIP".MARCHA_CIP_LINEA_2 AND "MARCA_SELECCION_L2_CIP" AND ((NOT "DETECTOR FLUJO RET_L2" AND NOT "MARCAS CIP".RUN_CIP_TANQUE_5 AND NOT "MARCAS CIP".RUN_CIP_TANQUE_6 AND NOT "MARCAS CIP".RUN_CIP_TANQUE_7 AND NOT "MARCAS CIP".RUN_CIP_TANQUE_8 AND NOT "MARCAS CIP".RUN_CIP_TANQUE_9 AND NOT "MARCAS CIP".RUN_CIP_TQ_QUESO_FLAN AND NOT "MARCAS CIP".RUN_CIP_TANQUE_14 AND NOT "MARCAS CIP".RUN_CIP_TANQUE_15 AND NOT "MARCAS CIP".RUN_CIP_TQ14_15_FLAN AND NOT "MARCAS CIP".RUN_CIP_FLAN_PAS2500 AND NOT "MARCAS CIP".RUN_CIP_TANQUE_10D AND NOT "MARCAS CIP".RUN_CIP_TANQUE_10E AND NOT "MARCAS CIP".RUN_CIP_INTERMEDIO_10D AND NOT "MARCAS CIP".RUN_CIP_INTERMEDIO_10E) OR ("MARCAS CIP".RUN_CIP_TANQUE_5 AND NOT "DETECTOR FLUJO RET_L2" AND NOT "NIVEL MIN TQ 5") OR ("MARCAS CIP".RUN_CIP_TANQUE_6 AND NOT "DETECTOR FLUJO RET_L2" AND NOT "NIVEL MIN TQ 6") OR ("MARCAS CIP".RUN_CIP_TANQUE_7 AND NOT "DETECTOR FLUJO RET_L2" AND NOT "NIVEL MIN TQ 7") OR ("MARCAS CIP".RUN_CIP_TANQUE_8 AND NOT "DETECTOR FLUJO RET_L2" AND NOT "NIVEL MIN TQ 8") OR ("MARCAS CIP".RUN_CIP_TANQUE_9 AND NOT "DETECTOR FLUJO RET_L2" AND NOT "NIVEL MIN TQ 9") OR ("MARCAS CIP".RUN_CIP_TQ_QUESO_FLAN AND NOT "DETECTOR FLUJO RET_L2") OR ("MARCAS CIP".RUN_CIP_TANQUE_14 AND NOT "DETECTOR FLUJO RET_L2" AND NOT "NIVEL MIN TQ 14") OR ("MARCAS CIP".RUN_CIP_TANQUE_15 AND NOT "DETECTOR FLUJO RET_L2" AND NOT "NIVEL MIN TQ 15") OR ("MARCAS CIP".RUN_CIP_TQ14_15_FLAN AND NOT "DETECTOR FLUJO RET_L2" AND NOT "NIVEL MIN TQ 18") OR ("MARCAS CIP".RUN_CIP_FLAN_PAS2500 AND NOT "DETECTOR FLUJO RET_L2" AND NOT "NIVEL MIN TQ 19") OR ("MARCAS CIP".RUN_CIP_TANQUE_10D AND NOT "DETECTOR FLUJO RET_L2" AND NOT "NIVEL MINIMO TQ10D") OR ("MARCAS CIP".RUN_CIP_TANQUE_10E AND NOT "DETECTOR FLUJO RET_L2" AND NOT "NIVEL MINIMO TQ10E") OR ("MARCAS CIP".RUN_CIP_INTERMEDIO_10D AND NOT "DETECTOR FLUJO RET_L2" AND NOT "NIVEL MINIMO TQ10D") OR ("MARCAS CIP".RUN_CIP_INTERMEDIO_10E AND NOT "DETECTOR FLUJO RET_L2" AND NOT "NIVEL MINIMO TQ10E")),
          operand := "Tag_774");
END_REGION

REGION Network 12
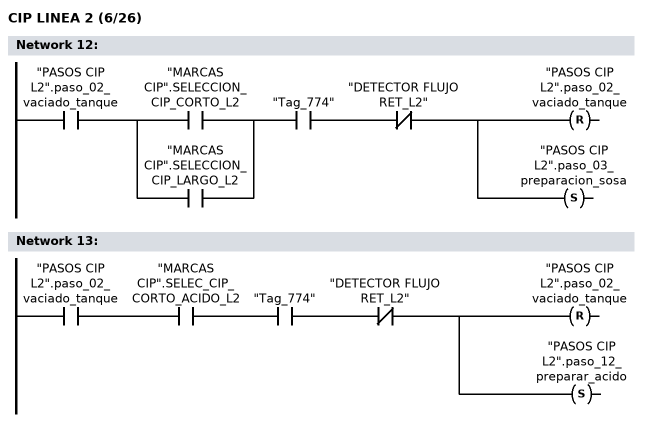
   RUNG wire#powerrail
      Contact( "PASOS CIP L2".paso_02_vaciado_tanque )
      wire#w1
      Contact( "MARCAS CIP".SELECCION_CIP_CORTO_L2 )
      wire#w2
      Contact( "Tag_774" )
      I_Contact( "DETECTOR FLUJO RET_L2" )
      wire#w3
      R_Coil( "PASOS CIP L2".paso_02_vaciado_tanque )
   END_RUNG
   RUNG wire#w1
      Contact( "MARCAS CIP".SELECCION_CIP_LARGO_L2 )
   END_RUNG wire#w2
   RUNG wire#w3
      S_Coil( "PASOS CIP L2".paso_03_preparacion_sosa )
   END_RUNG
   // the same network as SCL:
   #_w1 := "PASOS CIP L2".paso_02_vaciado_tanque AND ("MARCAS CIP".SELECCION_CIP_CORTO_L2 OR "MARCAS CIP".SELECCION_CIP_LARGO_L2) AND "Tag_774" AND NOT "DETECTOR FLUJO RET_L2";
   IF #_w1 THEN
       "PASOS CIP L2".paso_02_vaciado_tanque := FALSE;
       "PASOS CIP L2".paso_03_preparacion_sosa := TRUE;
   END_IF;
END_REGION

REGION Network 13
   RUNG wire#powerrail
      Contact( "PASOS CIP L2".paso_02_vaciado_tanque )
      Contact( "MARCAS CIP".SELEC_CIP_CORTO_ACIDO_L2 )
      Contact( "Tag_774" )
      I_Contact( "DETECTOR FLUJO RET_L2" )
      wire#w1
      R_Coil( "PASOS CIP L2".paso_02_vaciado_tanque )
   END_RUNG
   RUNG wire#w1
      S_Coil( "PASOS CIP L2".paso_12_preparar_acido )
   END_RUNG
   // the same network as SCL:
   #_w1 := "PASOS CIP L2".paso_02_vaciado_tanque AND "MARCAS CIP".SELEC_CIP_CORTO_ACIDO_L2 AND "Tag_774" AND NOT "DETECTOR FLUJO RET_L2";
   IF #_w1 THEN
       "PASOS CIP L2".paso_02_vaciado_tanque := FALSE;
       "PASOS CIP L2".paso_12_preparar_acido := TRUE;
   END_IF;
END_REGION

REGION Network 14
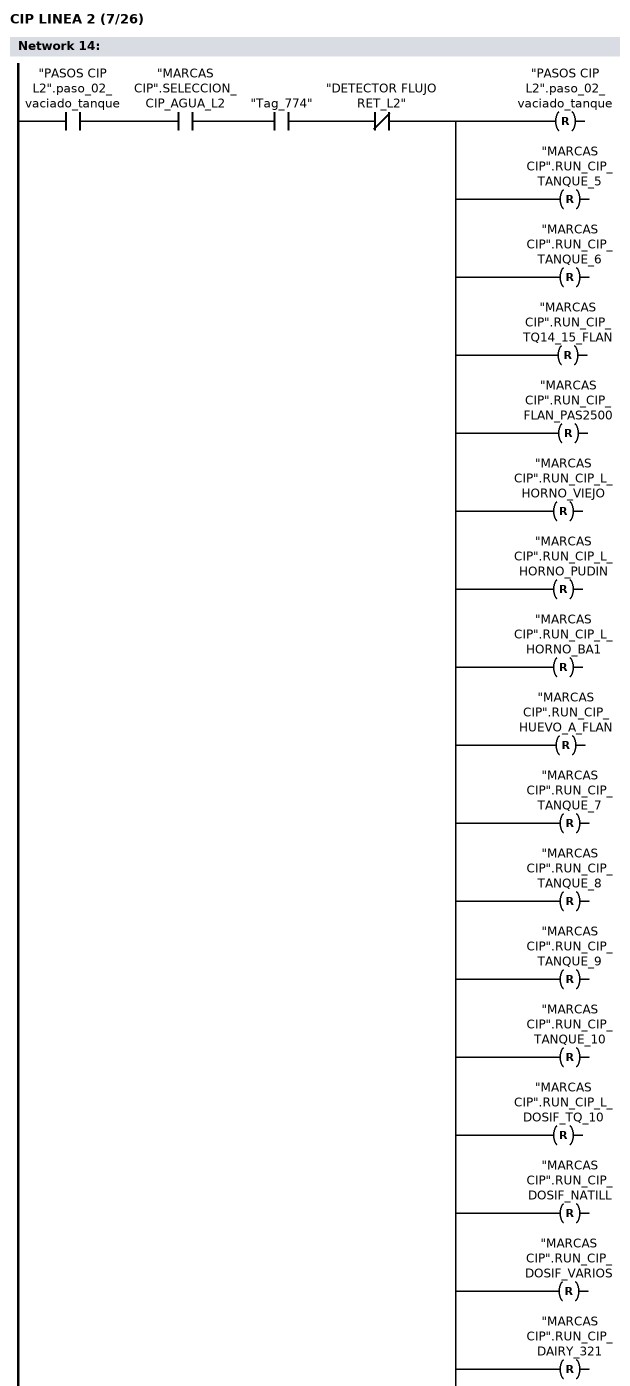
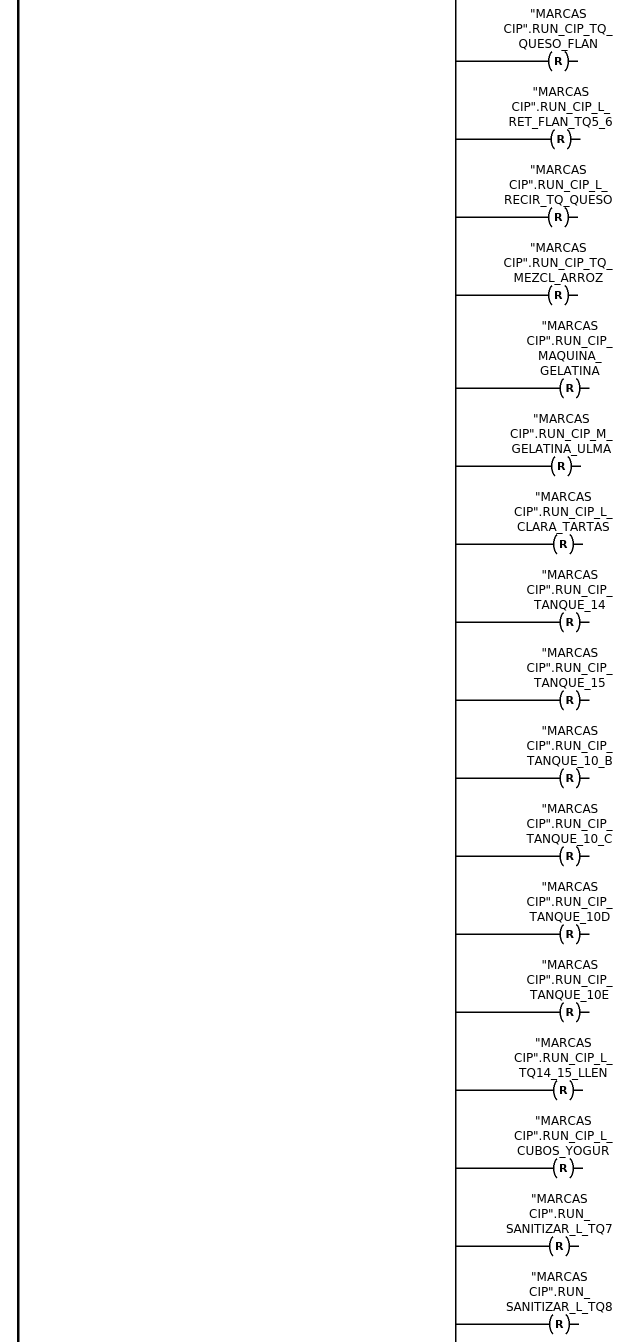
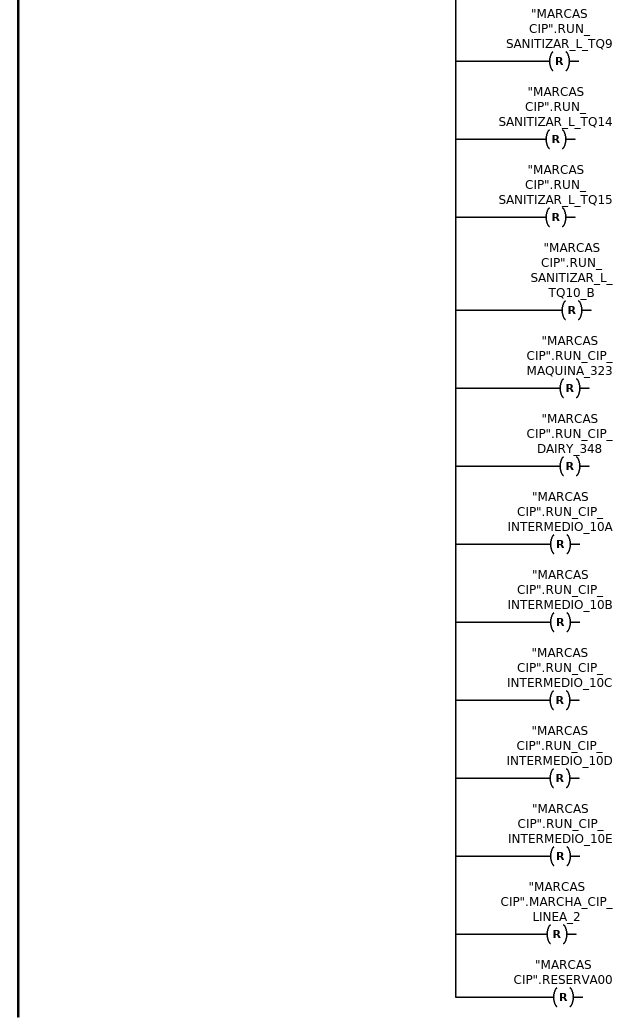
   RUNG wire#powerrail
      Contact( "PASOS CIP L2".paso_02_vaciado_tanque )
      Contact( "MARCAS CIP".SELECCION_CIP_AGUA_L2 )
      Contact( "Tag_774" )
      I_Contact( "DETECTOR FLUJO RET_L2" )
      wire#w1
      R_Coil( "PASOS CIP L2".paso_02_vaciado_tanque )
   END_RUNG
   RUNG wire#w1
      R_Coil( "MARCAS CIP".RUN_CIP_TANQUE_5 )
   END_RUNG
   RUNG wire#w1
      R_Coil( "MARCAS CIP".RUN_CIP_TANQUE_6 )
   END_RUNG
   RUNG wire#w1
      R_Coil( "MARCAS CIP".RUN_CIP_TQ14_15_FLAN )
   END_RUNG
   RUNG wire#w1
      R_Coil( "MARCAS CIP".RUN_CIP_FLAN_PAS2500 )
   END_RUNG
   RUNG wire#w1
      R_Coil( "MARCAS CIP".RUN_CIP_L_HORNO_VIEJO )
   END_RUNG
   RUNG wire#w1
      R_Coil( "MARCAS CIP".RUN_CIP_L_HORNO_PUDIN )
   END_RUNG
   RUNG wire#w1
      R_Coil( "MARCAS CIP".RUN_CIP_L_HORNO_BA1 )
   END_RUNG
   RUNG wire#w1
      R_Coil( "MARCAS CIP".RUN_CIP_HUEVO_A_FLAN )
   END_RUNG
   RUNG wire#w1
      R_Coil( "MARCAS CIP".RUN_CIP_TANQUE_7 )
   END_RUNG
   RUNG wire#w1
      R_Coil( "MARCAS CIP".RUN_CIP_TANQUE_8 )
   END_RUNG
   RUNG wire#w1
      R_Coil( "MARCAS CIP".RUN_CIP_TANQUE_9 )
   END_RUNG
   RUNG wire#w1
      R_Coil( "MARCAS CIP".RUN_CIP_TANQUE_10 )
   END_RUNG
   RUNG wire#w1
      R_Coil( "MARCAS CIP".RUN_CIP_L_DOSIF_TQ_10 )
   END_RUNG
   RUNG wire#w1
      R_Coil( "MARCAS CIP".RUN_CIP_DOSIF_NATILL )
   END_RUNG
   RUNG wire#w1
      R_Coil( "MARCAS CIP".RUN_CIP_DOSIF_VARIOS )
   END_RUNG
   RUNG wire#w1
      R_Coil( "MARCAS CIP".RUN_CIP_DAIRY_321 )
   END_RUNG
   RUNG wire#w1
      R_Coil( "MARCAS CIP".RUN_CIP_TQ_QUESO_FLAN )
   END_RUNG
   RUNG wire#w1
      R_Coil( "MARCAS CIP".RUN_CIP_L_RET_FLAN_TQ5_6 )
   END_RUNG
   RUNG wire#w1
      R_Coil( "MARCAS CIP".RUN_CIP_L_RECIR_TQ_QUESO )
   END_RUNG
   RUNG wire#w1
      R_Coil( "MARCAS CIP".RUN_CIP_TQ_MEZCL_ARROZ )
   END_RUNG
   RUNG wire#w1
      R_Coil( "MARCAS CIP".RUN_CIP_MAQUINA_GELATINA )
   END_RUNG
   RUNG wire#w1
      R_Coil( "MARCAS CIP".RUN_CIP_M_GELATINA_ULMA )
   END_RUNG
   RUNG wire#w1
      R_Coil( "MARCAS CIP".RUN_CIP_L_CLARA_TARTAS )
   END_RUNG
   RUNG wire#w1
      R_Coil( "MARCAS CIP".RUN_CIP_TANQUE_14 )
   END_RUNG
   RUNG wire#w1
      R_Coil( "MARCAS CIP".RUN_CIP_TANQUE_15 )
   END_RUNG
   RUNG wire#w1
      R_Coil( "MARCAS CIP".RUN_CIP_TANQUE_10_B )
   END_RUNG
   RUNG wire#w1
      R_Coil( "MARCAS CIP".RUN_CIP_TANQUE_10_C )
   END_RUNG
   RUNG wire#w1
      R_Coil( "MARCAS CIP".RUN_CIP_TANQUE_10D )
   END_RUNG
   RUNG wire#w1
      R_Coil( "MARCAS CIP".RUN_CIP_TANQUE_10E )
   END_RUNG
   RUNG wire#w1
      R_Coil( "MARCAS CIP".RUN_CIP_L_TQ14_15_LLEN )
   END_RUNG
   RUNG wire#w1
      R_Coil( "MARCAS CIP".RUN_CIP_L_CUBOS_YOGUR )
   END_RUNG
   RUNG wire#w1
      R_Coil( "MARCAS CIP".RUN_SANITIZAR_L_TQ7 )
   END_RUNG
   RUNG wire#w1
      R_Coil( "MARCAS CIP".RUN_SANITIZAR_L_TQ8 )
   END_RUNG
   RUNG wire#w1
      R_Coil( "MARCAS CIP".RUN_SANITIZAR_L_TQ9 )
   END_RUNG
   RUNG wire#w1
      R_Coil( "MARCAS CIP".RUN_SANITIZAR_L_TQ14 )
   END_RUNG
   RUNG wire#w1
      R_Coil( "MARCAS CIP".RUN_SANITIZAR_L_TQ15 )
   END_RUNG
   RUNG wire#w1
      R_Coil( "MARCAS CIP".RUN_SANITIZAR_L_TQ10_B )
   END_RUNG
   RUNG wire#w1
      R_Coil( "MARCAS CIP".RUN_CIP_MAQUINA_323 )
   END_RUNG
   RUNG wire#w1
      R_Coil( "MARCAS CIP".RUN_CIP_DAIRY_348 )
   END_RUNG
   RUNG wire#w1
      R_Coil( "MARCAS CIP".RUN_CIP_INTERMEDIO_10A )
   END_RUNG
   RUNG wire#w1
      R_Coil( "MARCAS CIP".RUN_CIP_INTERMEDIO_10B )
   END_RUNG
   RUNG wire#w1
      R_Coil( "MARCAS CIP".RUN_CIP_INTERMEDIO_10C )
   END_RUNG
   RUNG wire#w1
      R_Coil( "MARCAS CIP".RUN_CIP_INTERMEDIO_10D )
   END_RUNG
   RUNG wire#w1
      R_Coil( "MARCAS CIP".RUN_CIP_INTERMEDIO_10E )
   END_RUNG
   RUNG wire#w1
      R_Coil( "MARCAS CIP".MARCHA_CIP_LINEA_2 )
   END_RUNG
   RUNG wire#w1
      R_Coil( "MARCAS CIP".RESERVA00 )
   END_RUNG
   // the same network as SCL:
   #_w1 := "PASOS CIP L2".paso_02_vaciado_tanque AND "MARCAS CIP".SELECCION_CIP_AGUA_L2 AND "Tag_774" AND NOT "DETECTOR FLUJO RET_L2";
   IF #_w1 THEN
       "PASOS CIP L2".paso_02_vaciado_tanque := FALSE;
       "MARCAS CIP".RUN_CIP_TANQUE_5 := FALSE;
       "MARCAS CIP".RUN_CIP_TANQUE_6 := FALSE;
       "MARCAS CIP".RUN_CIP_TQ14_15_FLAN := FALSE;
       "MARCAS CIP".RUN_CIP_FLAN_PAS2500 := FALSE;
       "MARCAS CIP".RUN_CIP_L_HORNO_VIEJO := FALSE;
       "MARCAS CIP".RUN_CIP_L_HORNO_PUDIN := FALSE;
       "MARCAS CIP".RUN_CIP_L_HORNO_BA1 := FALSE;
       "MARCAS CIP".RUN_CIP_HUEVO_A_FLAN := FALSE;
       "MARCAS CIP".RUN_CIP_TANQUE_7 := FALSE;
       "MARCAS CIP".RUN_CIP_TANQUE_8 := FALSE;
       "MARCAS CIP".RUN_CIP_TANQUE_9 := FALSE;
       "MARCAS CIP".RUN_CIP_TANQUE_10 := FALSE;
       "MARCAS CIP".RUN_CIP_L_DOSIF_TQ_10 := FALSE;
       "MARCAS CIP".RUN_CIP_DOSIF_NATILL := FALSE;
       "MARCAS CIP".RUN_CIP_DOSIF_VARIOS := FALSE;
       "MARCAS CIP".RUN_CIP_DAIRY_321 := FALSE;
       "MARCAS CIP".RUN_CIP_TQ_QUESO_FLAN := FALSE;
       "MARCAS CIP".RUN_CIP_L_RET_FLAN_TQ5_6 := FALSE;
       "MARCAS CIP".RUN_CIP_L_RECIR_TQ_QUESO := FALSE;
       "MARCAS CIP".RUN_CIP_TQ_MEZCL_ARROZ := FALSE;
       "MARCAS CIP".RUN_CIP_MAQUINA_GELATINA := FALSE;
       "MARCAS CIP".RUN_CIP_M_GELATINA_ULMA := FALSE;
       "MARCAS CIP".RUN_CIP_L_CLARA_TARTAS := FALSE;
       "MARCAS CIP".RUN_CIP_TANQUE_14 := FALSE;
       "MARCAS CIP".RUN_CIP_TANQUE_15 := FALSE;
       "MARCAS CIP".RUN_CIP_TANQUE_10_B := FALSE;
       "MARCAS CIP".RUN_CIP_TANQUE_10_C := FALSE;
       "MARCAS CIP".RUN_CIP_TANQUE_10D := FALSE;
       "MARCAS CIP".RUN_CIP_TANQUE_10E := FALSE;
       "MARCAS CIP".RUN_CIP_L_TQ14_15_LLEN := FALSE;
       "MARCAS CIP".RUN_CIP_L_CUBOS_YOGUR := FALSE;
       "MARCAS CIP".RUN_SANITIZAR_L_TQ7 := FALSE;
       "MARCAS CIP".RUN_SANITIZAR_L_TQ8 := FALSE;
       "MARCAS CIP".RUN_SANITIZAR_L_TQ9 := FALSE;
       "MARCAS CIP".RUN_SANITIZAR_L_TQ14 := FALSE;
       "MARCAS CIP".RUN_SANITIZAR_L_TQ15 := FALSE;
       "MARCAS CIP".RUN_SANITIZAR_L_TQ10_B := FALSE;
       "MARCAS CIP".RUN_CIP_MAQUINA_323 := FALSE;
       "MARCAS CIP".RUN_CIP_DAIRY_348 := FALSE;
       "MARCAS CIP".RUN_CIP_INTERMEDIO_10A := FALSE;
       "MARCAS CIP".RUN_CIP_INTERMEDIO_10B := FALSE;
       "MARCAS CIP".RUN_CIP_INTERMEDIO_10C := FALSE;
       "MARCAS CIP".RUN_CIP_INTERMEDIO_10D := FALSE;
       "MARCAS CIP".RUN_CIP_INTERMEDIO_10E := FALSE;
       "MARCAS CIP".MARCHA_CIP_LINEA_2 := FALSE;
       "MARCAS CIP".RESERVA00 := FALSE;
   END_IF;
END_REGION

REGION Network 15
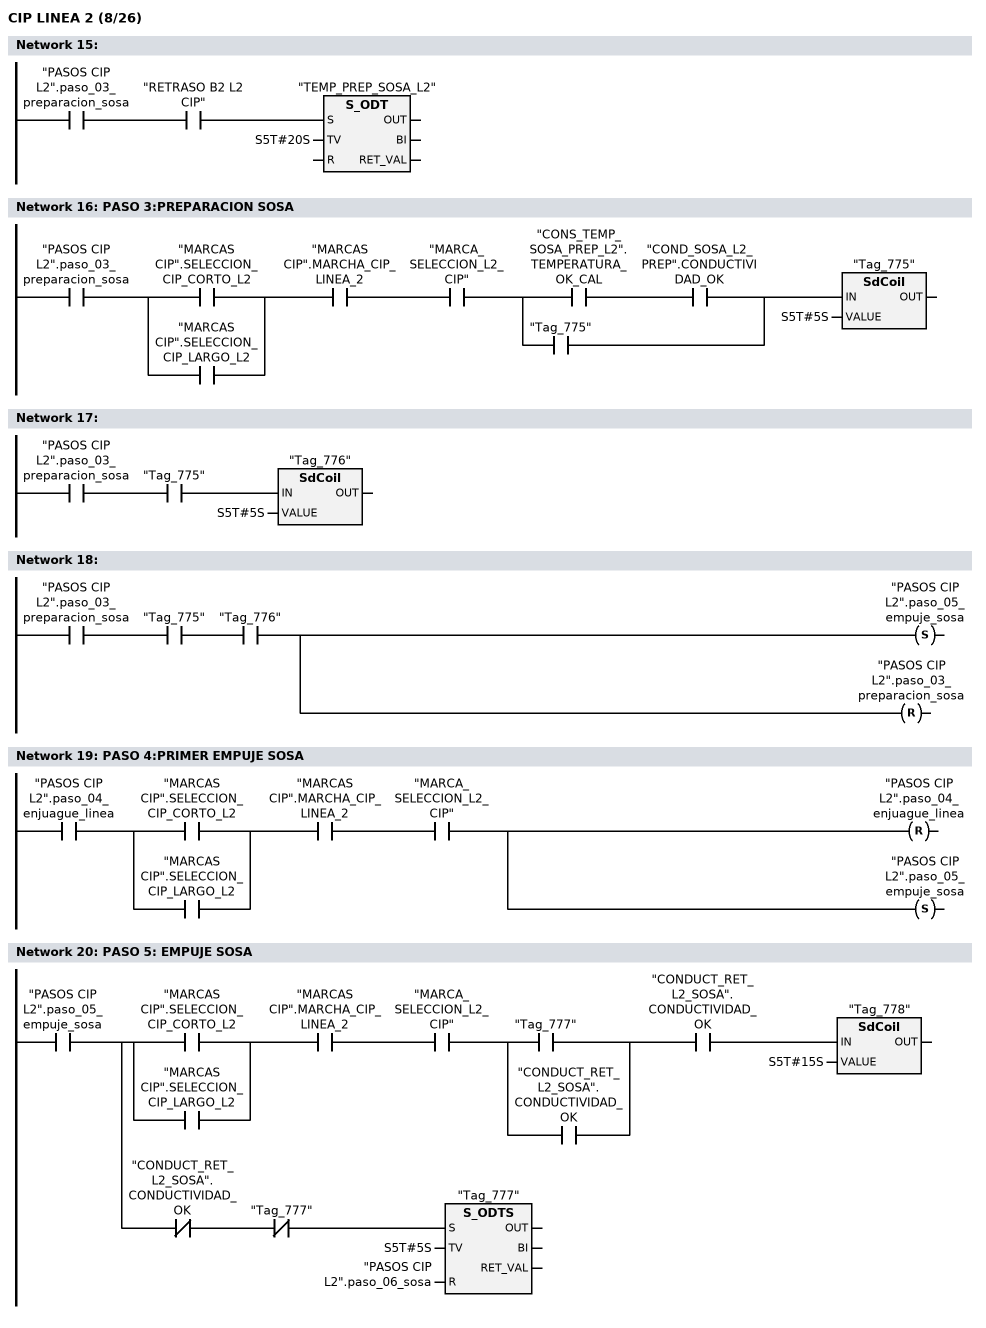
   RUNG wire#powerrail
      Contact( "PASOS CIP L2".paso_03_preparacion_sosa )
      Contact( "RETRASO B2 L2 CIP" )
      S_ODT(T_NO := "TEMP_PREP_SOSA_L2", TV := S5T#20S, R :=, BI =>, RET_VAL =>)
   END_RUNG
   // the same network as SCL:
   #_s5time1 := S_ODT(T_NO := "TEMP_PREP_SOSA_L2",
                      TV := S5T#20S,
                      S := "PASOS CIP L2".paso_03_preparacion_sosa AND "RETRASO B2 L2 CIP");
END_REGION

REGION Network 16: PASO 3:PREPARACION SOSA
   // no SCL statement known for SdCoil: written as a call
   SdCoil(value := S5T#5S,
          in := "PASOS CIP L2".paso_03_preparacion_sosa AND ("MARCAS CIP".SELECCION_CIP_CORTO_L2 OR "MARCAS CIP".SELECCION_CIP_LARGO_L2) AND "MARCAS CIP".MARCHA_CIP_LINEA_2 AND "MARCA_SELECCION_L2_CIP" AND (("CONS_TEMP_SOSA_PREP_L2".TEMPERATURA_OK_CAL AND "COND_SOSA_L2_PREP".CONDUCTIVIDAD_OK) OR "Tag_775"),
          operand := "Tag_775");
END_REGION

REGION Network 17
   // no SCL statement known for SdCoil: written as a call
   SdCoil(value := S5T#5S, operand := "Tag_776", in := "PASOS CIP L2".paso_03_preparacion_sosa AND "Tag_775");
END_REGION

REGION Network 18
   RUNG wire#powerrail
      Contact( "PASOS CIP L2".paso_03_preparacion_sosa )
      Contact( "Tag_775" )
      Contact( "Tag_776" )
      wire#w1
      S_Coil( "PASOS CIP L2".paso_05_empuje_sosa )
   END_RUNG
   RUNG wire#w1
      R_Coil( "PASOS CIP L2".paso_03_preparacion_sosa )
   END_RUNG
   // the same network as SCL:
   IF "PASOS CIP L2".paso_03_preparacion_sosa AND "Tag_775" AND "Tag_776" THEN
       "PASOS CIP L2".paso_05_empuje_sosa := TRUE;
       "PASOS CIP L2".paso_03_preparacion_sosa := FALSE;
   END_IF;
END_REGION

REGION Network 19: PASO 4:PRIMER EMPUJE SOSA
   RUNG wire#powerrail
      Contact( "PASOS CIP L2".paso_04_enjuague_linea )
      wire#w1
      Contact( "MARCAS CIP".SELECCION_CIP_CORTO_L2 )
      wire#w2
      Contact( "MARCAS CIP".MARCHA_CIP_LINEA_2 )
      Contact( "MARCA_SELECCION_L2_CIP" )
      wire#w3
      R_Coil( "PASOS CIP L2".paso_04_enjuague_linea )
   END_RUNG
   RUNG wire#w1
      Contact( "MARCAS CIP".SELECCION_CIP_LARGO_L2 )
   END_RUNG wire#w2
   RUNG wire#w3
      S_Coil( "PASOS CIP L2".paso_05_empuje_sosa )
   END_RUNG
   // the same network as SCL:
   #_w1 := "PASOS CIP L2".paso_04_enjuague_linea AND ("MARCAS CIP".SELECCION_CIP_CORTO_L2 OR "MARCAS CIP".SELECCION_CIP_LARGO_L2) AND "MARCAS CIP".MARCHA_CIP_LINEA_2 AND "MARCA_SELECCION_L2_CIP";
   IF #_w1 THEN
       "PASOS CIP L2".paso_04_enjuague_linea := FALSE;
       "PASOS CIP L2".paso_05_empuje_sosa := TRUE;
   END_IF;
END_REGION

REGION Network 20: PASO 5: EMPUJE SOSA
   // no SCL statement known for SdCoil: written as a call
   #_w1 := "PASOS CIP L2".paso_05_empuje_sosa;
   SdCoil(value := S5T#15S,
          operand := "Tag_778",
          in := "PASOS CIP L2".paso_05_empuje_sosa AND ("MARCAS CIP".SELECCION_CIP_CORTO_L2 OR "MARCAS CIP".SELECCION_CIP_LARGO_L2) AND "MARCAS CIP".MARCHA_CIP_LINEA_2 AND "MARCA_SELECCION_L2_CIP" AND ("Tag_777" OR "CONDUCT_RET_L2_SOSA".CONDUCTIVIDAD_OK) AND "CONDUCT_RET_L2_SOSA".CONDUCTIVIDAD_OK);
   #_s5time1 := S_ODTS(T_NO := "Tag_777",
                       TV := S5T#5S,
                       R := "PASOS CIP L2".paso_06_sosa,
                       S := #_w1 AND NOT "CONDUCT_RET_L2_SOSA".CONDUCTIVIDAD_OK AND NOT "Tag_777");
END_REGION

REGION Network 21
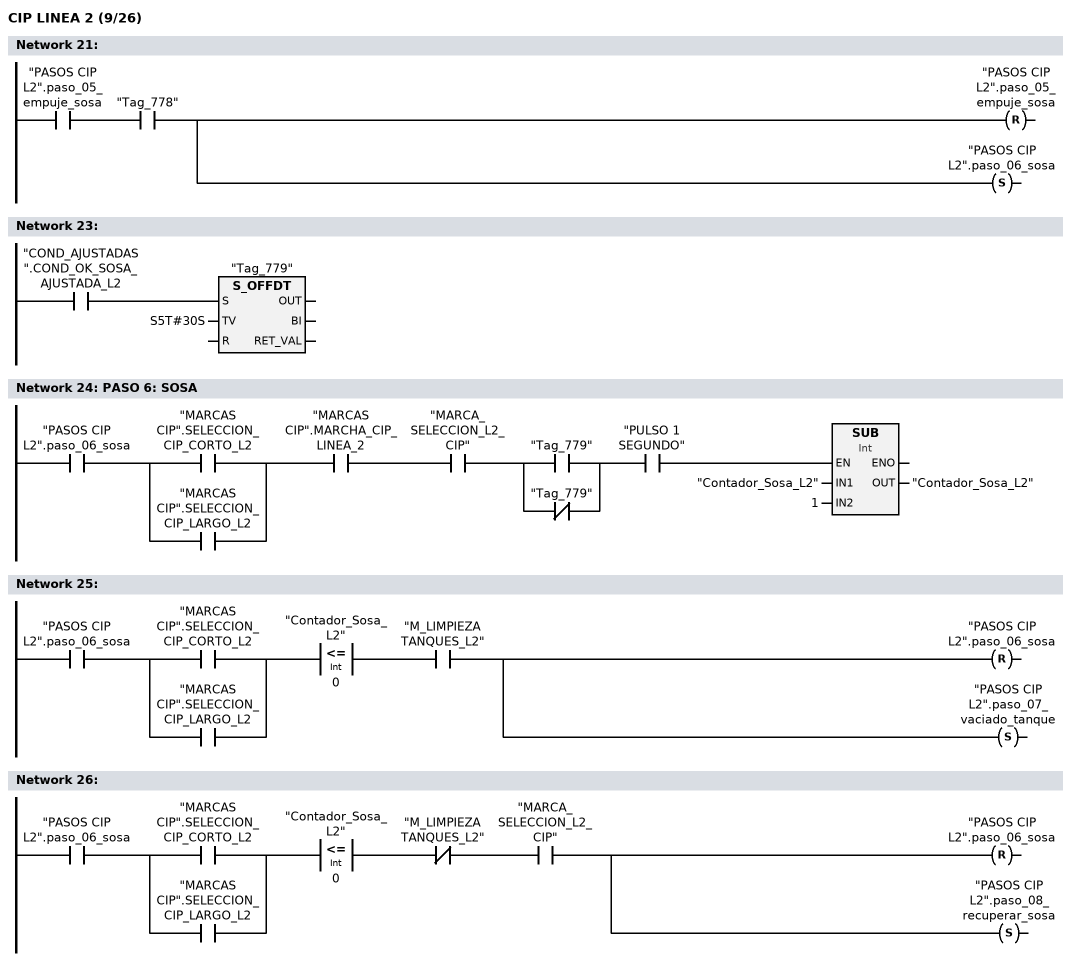
   RUNG wire#powerrail
      Contact( "PASOS CIP L2".paso_05_empuje_sosa )
      Contact( "Tag_778" )
      wire#w1
      R_Coil( "PASOS CIP L2".paso_05_empuje_sosa )
   END_RUNG
   RUNG wire#w1
      S_Coil( "PASOS CIP L2".paso_06_sosa )
   END_RUNG
   // the same network as SCL:
   #_w1 := "PASOS CIP L2".paso_05_empuje_sosa AND "Tag_778";
   IF #_w1 THEN
       "PASOS CIP L2".paso_05_empuje_sosa := FALSE;
       "PASOS CIP L2".paso_06_sosa := TRUE;
   END_IF;
END_REGION

NETWORK
TITLE = 
      A     "PASOS CIP L2".paso_06_sosa;
      JC    c1;
      L     "SP TIM L2 CIP".TIM_PASO_6_L2;
      L     60;
      *I;
      T     "Contador_Sosa_L2";
c1:   NOP   0;

REGION Network 23
   RUNG wire#powerrail
      Contact( "COND_AJUSTADAS".COND_OK_SOSA_AJUSTADA_L2 )
      S_OFFDT(T_NO := "Tag_779", TV := S5T#30S, R :=, BI =>, RET_VAL =>)
   END_RUNG
   // the same network as SCL:
   #_s5time1 := S_OFFDT(T_NO := "Tag_779", TV := S5T#30S, S := "COND_AJUSTADAS".COND_OK_SOSA_AJUSTADA_L2);
END_REGION

REGION Network 24: PASO 6: SOSA
   RUNG wire#powerrail
      Contact( "PASOS CIP L2".paso_06_sosa )
      wire#w1
      Contact( "MARCAS CIP".SELECCION_CIP_CORTO_L2 )
      wire#w2
      Contact( "MARCAS CIP".MARCHA_CIP_LINEA_2 )
      Contact( "MARCA_SELECCION_L2_CIP" )
      wire#w3
      Contact( "Tag_779" )
      wire#w4
      Contact( "PULSO 1 SEGUNDO" )
      { S7_Templates := "SrcType := Int"; S7_GenerateENO := "TRUE" } Sub(in1 := "Contador_Sosa_L2", in2 := 1, out => "Contador_Sosa_L2")
   END_RUNG
   RUNG wire#w1
      Contact( "MARCAS CIP".SELECCION_CIP_LARGO_L2 )
   END_RUNG wire#w2
   RUNG wire#w3
      I_Contact( "Tag_779" )
   END_RUNG wire#w4
   // the same network as SCL:
   IF "PASOS CIP L2".paso_06_sosa AND ("MARCAS CIP".SELECCION_CIP_CORTO_L2 OR "MARCAS CIP".SELECCION_CIP_LARGO_L2) AND "MARCAS CIP".MARCHA_CIP_LINEA_2 AND "MARCA_SELECCION_L2_CIP" AND ("Tag_779" OR NOT "Tag_779") AND "PULSO 1 SEGUNDO" THEN
       "Contador_Sosa_L2" := "Contador_Sosa_L2" - 1;
   END_IF;
END_REGION

REGION Network 25
   RUNG wire#powerrail
      Contact( "PASOS CIP L2".paso_06_sosa )
      wire#w1
      Contact( "MARCAS CIP".SELECCION_CIP_CORTO_L2 )
      wire#w2
      { S7_Templates := "SrcType := Int" } LE_Contact(in1 := "Contador_Sosa_L2", in2 := 0)
      Contact( "M_LIMPIEZA TANQUES_L2" )
      wire#w3
      R_Coil( "PASOS CIP L2".paso_06_sosa )
   END_RUNG
   RUNG wire#w1
      Contact( "MARCAS CIP".SELECCION_CIP_LARGO_L2 )
   END_RUNG wire#w2
   RUNG wire#w3
      S_Coil( "PASOS CIP L2".paso_07_vaciado_tanque )
   END_RUNG
   // the same network as SCL:
   #_w1 := "PASOS CIP L2".paso_06_sosa AND ("MARCAS CIP".SELECCION_CIP_CORTO_L2 OR "MARCAS CIP".SELECCION_CIP_LARGO_L2) AND ("Contador_Sosa_L2" <= 0) AND "M_LIMPIEZA TANQUES_L2";
   IF #_w1 THEN
       "PASOS CIP L2".paso_06_sosa := FALSE;
       "PASOS CIP L2".paso_07_vaciado_tanque := TRUE;
   END_IF;
END_REGION

REGION Network 26
   RUNG wire#powerrail
      Contact( "PASOS CIP L2".paso_06_sosa )
      wire#w1
      Contact( "MARCAS CIP".SELECCION_CIP_CORTO_L2 )
      wire#w2
      { S7_Templates := "SrcType := Int" } LE_Contact(in1 := "Contador_Sosa_L2", in2 := 0)
      I_Contact( "M_LIMPIEZA TANQUES_L2" )
      Contact( "MARCA_SELECCION_L2_CIP" )
      wire#w3
      R_Coil( "PASOS CIP L2".paso_06_sosa )
   END_RUNG
   RUNG wire#w1
      Contact( "MARCAS CIP".SELECCION_CIP_LARGO_L2 )
   END_RUNG wire#w2
   RUNG wire#w3
      S_Coil( "PASOS CIP L2".paso_08_recuperar_sosa )
   END_RUNG
   // the same network as SCL:
   #_w1 := "PASOS CIP L2".paso_06_sosa AND ("MARCAS CIP".SELECCION_CIP_CORTO_L2 OR "MARCAS CIP".SELECCION_CIP_LARGO_L2) AND ("Contador_Sosa_L2" <= 0) AND NOT "M_LIMPIEZA TANQUES_L2" AND "MARCA_SELECCION_L2_CIP";
   IF #_w1 THEN
       "PASOS CIP L2".paso_06_sosa := FALSE;
       "PASOS CIP L2".paso_08_recuperar_sosa := TRUE;
   END_IF;
END_REGION

REGION Network 27: PASO 7: VACIADO SI TANQUE
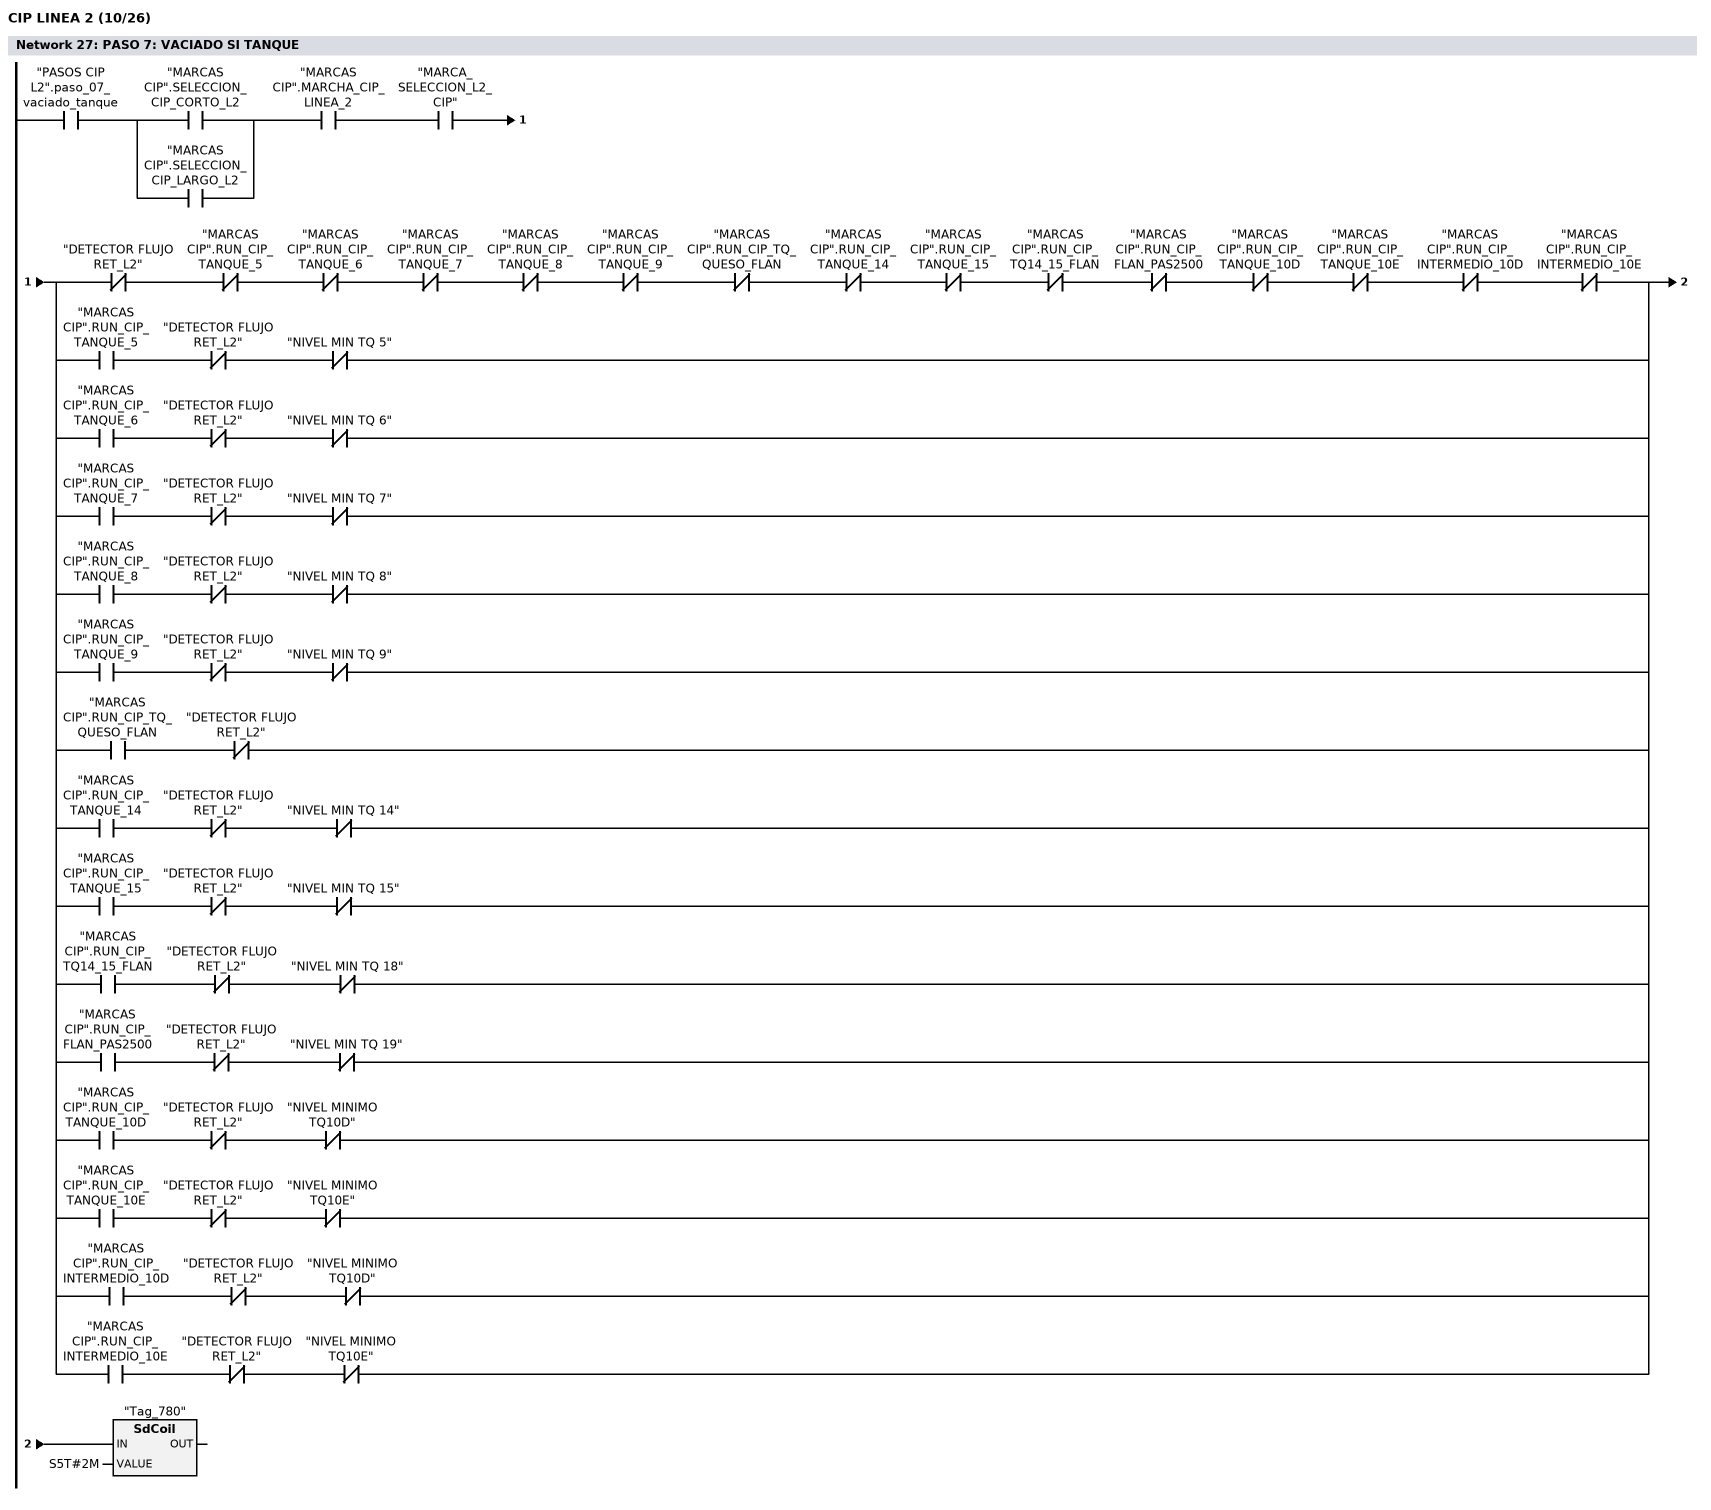
   // no SCL statement known for SdCoil: written as a call
   SdCoil(value := S5T#2M,
          in := "PASOS CIP L2".paso_07_vaciado_tanque AND ("MARCAS CIP".SELECCION_CIP_CORTO_L2 OR "MARCAS CIP".SELECCION_CIP_LARGO_L2) AND "MARCAS CIP".MARCHA_CIP_LINEA_2 AND "MARCA_SELECCION_L2_CIP" AND ((NOT "DETECTOR FLUJO RET_L2" AND NOT "MARCAS CIP".RUN_CIP_TANQUE_5 AND NOT "MARCAS CIP".RUN_CIP_TANQUE_6 AND NOT "MARCAS CIP".RUN_CIP_TANQUE_7 AND NOT "MARCAS CIP".RUN_CIP_TANQUE_8 AND NOT "MARCAS CIP".RUN_CIP_TANQUE_9 AND NOT "MARCAS CIP".RUN_CIP_TQ_QUESO_FLAN AND NOT "MARCAS CIP".RUN_CIP_TANQUE_14 AND NOT "MARCAS CIP".RUN_CIP_TANQUE_15 AND NOT "MARCAS CIP".RUN_CIP_TQ14_15_FLAN AND NOT "MARCAS CIP".RUN_CIP_FLAN_PAS2500 AND NOT "MARCAS CIP".RUN_CIP_TANQUE_10D AND NOT "MARCAS CIP".RUN_CIP_TANQUE_10E AND NOT "MARCAS CIP".RUN_CIP_INTERMEDIO_10D AND NOT "MARCAS CIP".RUN_CIP_INTERMEDIO_10E) OR ("MARCAS CIP".RUN_CIP_TANQUE_5 AND NOT "DETECTOR FLUJO RET_L2" AND NOT "NIVEL MIN TQ 5") OR ("MARCAS CIP".RUN_CIP_TANQUE_6 AND NOT "DETECTOR FLUJO RET_L2" AND NOT "NIVEL MIN TQ 6") OR ("MARCAS CIP".RUN_CIP_TANQUE_7 AND NOT "DETECTOR FLUJO RET_L2" AND NOT "NIVEL MIN TQ 7") OR ("MARCAS CIP".RUN_CIP_TANQUE_8 AND NOT "DETECTOR FLUJO RET_L2" AND NOT "NIVEL MIN TQ 8") OR ("MARCAS CIP".RUN_CIP_TANQUE_9 AND NOT "DETECTOR FLUJO RET_L2" AND NOT "NIVEL MIN TQ 9") OR ("MARCAS CIP".RUN_CIP_TQ_QUESO_FLAN AND NOT "DETECTOR FLUJO RET_L2") OR ("MARCAS CIP".RUN_CIP_TANQUE_14 AND NOT "DETECTOR FLUJO RET_L2" AND NOT "NIVEL MIN TQ 14") OR ("MARCAS CIP".RUN_CIP_TANQUE_15 AND NOT "DETECTOR FLUJO RET_L2" AND NOT "NIVEL MIN TQ 15") OR ("MARCAS CIP".RUN_CIP_TQ14_15_FLAN AND NOT "DETECTOR FLUJO RET_L2" AND NOT "NIVEL MIN TQ 18") OR ("MARCAS CIP".RUN_CIP_FLAN_PAS2500 AND NOT "DETECTOR FLUJO RET_L2" AND NOT "NIVEL MIN TQ 19") OR ("MARCAS CIP".RUN_CIP_TANQUE_10D AND NOT "DETECTOR FLUJO RET_L2" AND NOT "NIVEL MINIMO TQ10D") OR ("MARCAS CIP".RUN_CIP_TANQUE_10E AND NOT "DETECTOR FLUJO RET_L2" AND NOT "NIVEL MINIMO TQ10E") OR ("MARCAS CIP".RUN_CIP_INTERMEDIO_10D AND NOT "DETECTOR FLUJO RET_L2" AND NOT "NIVEL MINIMO TQ10D") OR ("MARCAS CIP".RUN_CIP_INTERMEDIO_10E AND NOT "DETECTOR FLUJO RET_L2" AND NOT "NIVEL MINIMO TQ10E")),
          operand := "Tag_780");
END_REGION

REGION Network 28
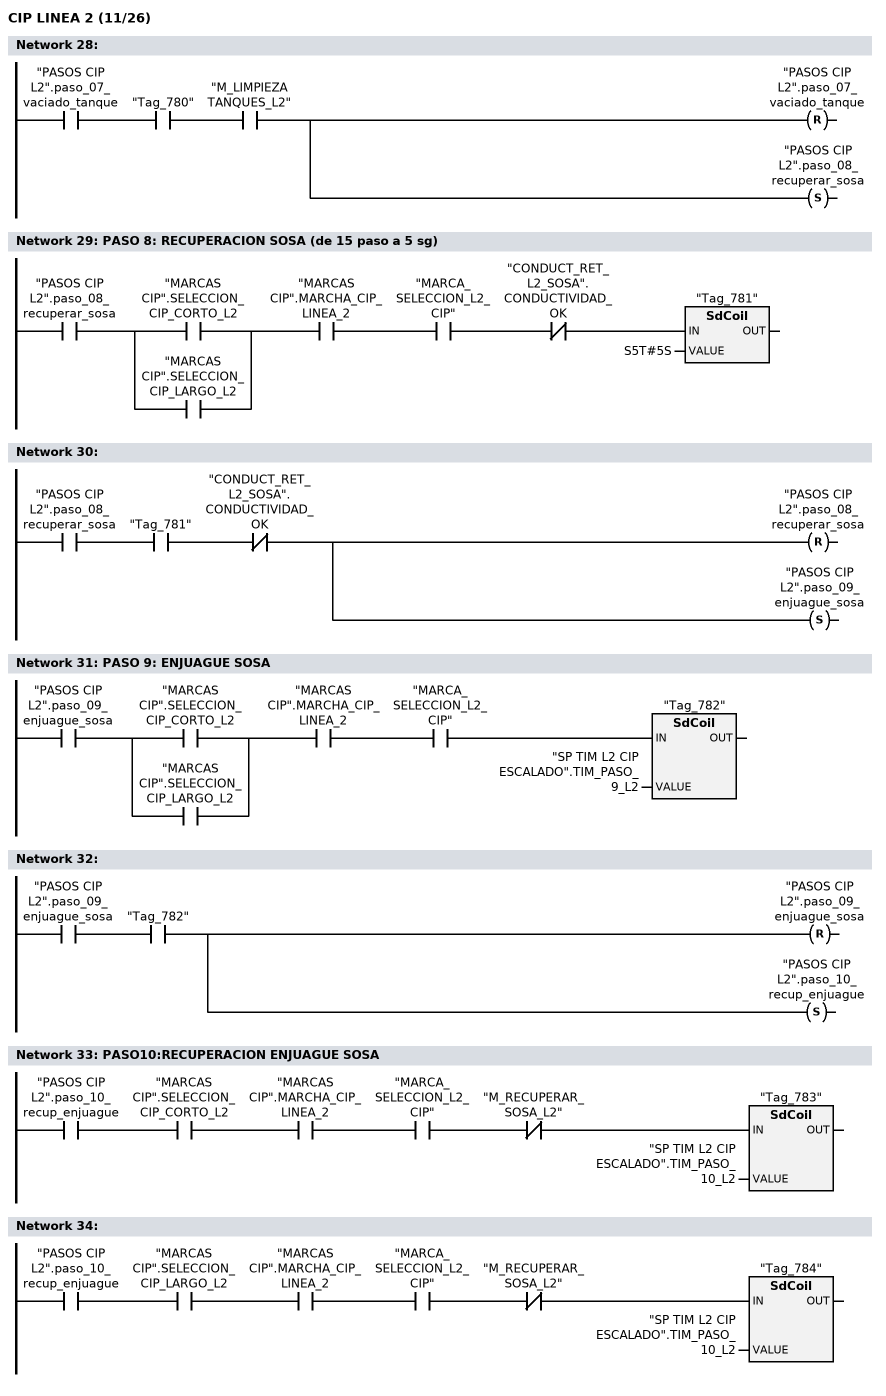
   RUNG wire#powerrail
      Contact( "PASOS CIP L2".paso_07_vaciado_tanque )
      Contact( "Tag_780" )
      Contact( "M_LIMPIEZA TANQUES_L2" )
      wire#w1
      R_Coil( "PASOS CIP L2".paso_07_vaciado_tanque )
   END_RUNG
   RUNG wire#w1
      S_Coil( "PASOS CIP L2".paso_08_recuperar_sosa )
   END_RUNG
   // the same network as SCL:
   #_w1 := "PASOS CIP L2".paso_07_vaciado_tanque AND "Tag_780" AND "M_LIMPIEZA TANQUES_L2";
   IF #_w1 THEN
       "PASOS CIP L2".paso_07_vaciado_tanque := FALSE;
       "PASOS CIP L2".paso_08_recuperar_sosa := TRUE;
   END_IF;
END_REGION

REGION Network 29: PASO 8: RECUPERACION SOSA (de 15 paso a 5 sg)
   // no SCL statement known for SdCoil: written as a call
   SdCoil(value := S5T#5S,
          operand := "Tag_781",
          in := "PASOS CIP L2".paso_08_recuperar_sosa AND ("MARCAS CIP".SELECCION_CIP_CORTO_L2 OR "MARCAS CIP".SELECCION_CIP_LARGO_L2) AND "MARCAS CIP".MARCHA_CIP_LINEA_2 AND "MARCA_SELECCION_L2_CIP" AND NOT "CONDUCT_RET_L2_SOSA".CONDUCTIVIDAD_OK);
END_REGION

REGION Network 30
   RUNG wire#powerrail
      Contact( "PASOS CIP L2".paso_08_recuperar_sosa )
      Contact( "Tag_781" )
      I_Contact( "CONDUCT_RET_L2_SOSA".CONDUCTIVIDAD_OK )
      wire#w1
      R_Coil( "PASOS CIP L2".paso_08_recuperar_sosa )
   END_RUNG
   RUNG wire#w1
      S_Coil( "PASOS CIP L2".paso_09_enjuague_sosa )
   END_RUNG
   // the same network as SCL:
   #_w1 := "PASOS CIP L2".paso_08_recuperar_sosa AND "Tag_781" AND NOT "CONDUCT_RET_L2_SOSA".CONDUCTIVIDAD_OK;
   IF #_w1 THEN
       "PASOS CIP L2".paso_08_recuperar_sosa := FALSE;
       "PASOS CIP L2".paso_09_enjuague_sosa := TRUE;
   END_IF;
END_REGION

REGION Network 31: PASO 9: ENJUAGUE SOSA
   // no SCL statement known for SdCoil: written as a call
   SdCoil(value := "SP TIM L2 CIP ESCALADO".TIM_PASO_9_L2,
          operand := "Tag_782",
          in := "PASOS CIP L2".paso_09_enjuague_sosa AND ("MARCAS CIP".SELECCION_CIP_CORTO_L2 OR "MARCAS CIP".SELECCION_CIP_LARGO_L2) AND "MARCAS CIP".MARCHA_CIP_LINEA_2 AND "MARCA_SELECCION_L2_CIP");
END_REGION

REGION Network 32
   RUNG wire#powerrail
      Contact( "PASOS CIP L2".paso_09_enjuague_sosa )
      Contact( "Tag_782" )
      wire#w1
      R_Coil( "PASOS CIP L2".paso_09_enjuague_sosa )
   END_RUNG
   RUNG wire#w1
      S_Coil( "PASOS CIP L2".paso_10_recup_enjuague )
   END_RUNG
   // the same network as SCL:
   #_w1 := "PASOS CIP L2".paso_09_enjuague_sosa AND "Tag_782";
   IF #_w1 THEN
       "PASOS CIP L2".paso_09_enjuague_sosa := FALSE;
       "PASOS CIP L2".paso_10_recup_enjuague := TRUE;
   END_IF;
END_REGION

REGION Network 33: PASO10:RECUPERACION ENJUAGUE SOSA
   // no SCL statement known for SdCoil: written as a call
   SdCoil(value := "SP TIM L2 CIP ESCALADO".TIM_PASO_10_L2,
          operand := "Tag_783",
          in := "PASOS CIP L2".paso_10_recup_enjuague AND "MARCAS CIP".SELECCION_CIP_CORTO_L2 AND "MARCAS CIP".MARCHA_CIP_LINEA_2 AND "MARCA_SELECCION_L2_CIP" AND NOT "M_RECUPERAR_SOSA_L2");
END_REGION

REGION Network 34
   // no SCL statement known for SdCoil: written as a call
   SdCoil(value := "SP TIM L2 CIP ESCALADO".TIM_PASO_10_L2,
          operand := "Tag_784",
          in := "PASOS CIP L2".paso_10_recup_enjuague AND "MARCAS CIP".SELECCION_CIP_LARGO_L2 AND "MARCAS CIP".MARCHA_CIP_LINEA_2 AND "MARCA_SELECCION_L2_CIP" AND NOT "M_RECUPERAR_SOSA_L2");
END_REGION

REGION Network 35
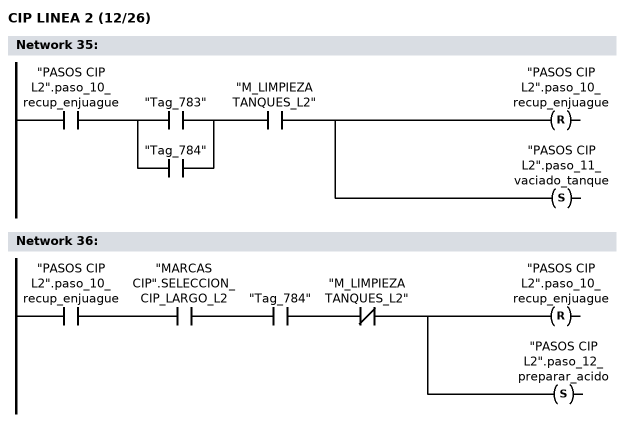
   RUNG wire#powerrail
      Contact( "PASOS CIP L2".paso_10_recup_enjuague )
      wire#w1
      Contact( "Tag_783" )
      wire#w2
      Contact( "M_LIMPIEZA TANQUES_L2" )
      wire#w3
      R_Coil( "PASOS CIP L2".paso_10_recup_enjuague )
   END_RUNG
   RUNG wire#w1
      Contact( "Tag_784" )
   END_RUNG wire#w2
   RUNG wire#w3
      S_Coil( "PASOS CIP L2".paso_11_vaciado_tanque )
   END_RUNG
   // the same network as SCL:
   #_w1 := "PASOS CIP L2".paso_10_recup_enjuague AND ("Tag_783" OR "Tag_784") AND "M_LIMPIEZA TANQUES_L2";
   IF #_w1 THEN
       "PASOS CIP L2".paso_10_recup_enjuague := FALSE;
       "PASOS CIP L2".paso_11_vaciado_tanque := TRUE;
   END_IF;
END_REGION

REGION Network 36
   RUNG wire#powerrail
      Contact( "PASOS CIP L2".paso_10_recup_enjuague )
      Contact( "MARCAS CIP".SELECCION_CIP_LARGO_L2 )
      Contact( "Tag_784" )
      I_Contact( "M_LIMPIEZA TANQUES_L2" )
      wire#w1
      R_Coil( "PASOS CIP L2".paso_10_recup_enjuague )
   END_RUNG
   RUNG wire#w1
      S_Coil( "PASOS CIP L2".paso_12_preparar_acido )
   END_RUNG
   // the same network as SCL:
   #_w1 := "PASOS CIP L2".paso_10_recup_enjuague AND "MARCAS CIP".SELECCION_CIP_LARGO_L2 AND "Tag_784" AND NOT "M_LIMPIEZA TANQUES_L2";
   IF #_w1 THEN
       "PASOS CIP L2".paso_10_recup_enjuague := FALSE;
       "PASOS CIP L2".paso_12_preparar_acido := TRUE;
   END_IF;
END_REGION

REGION Network 37
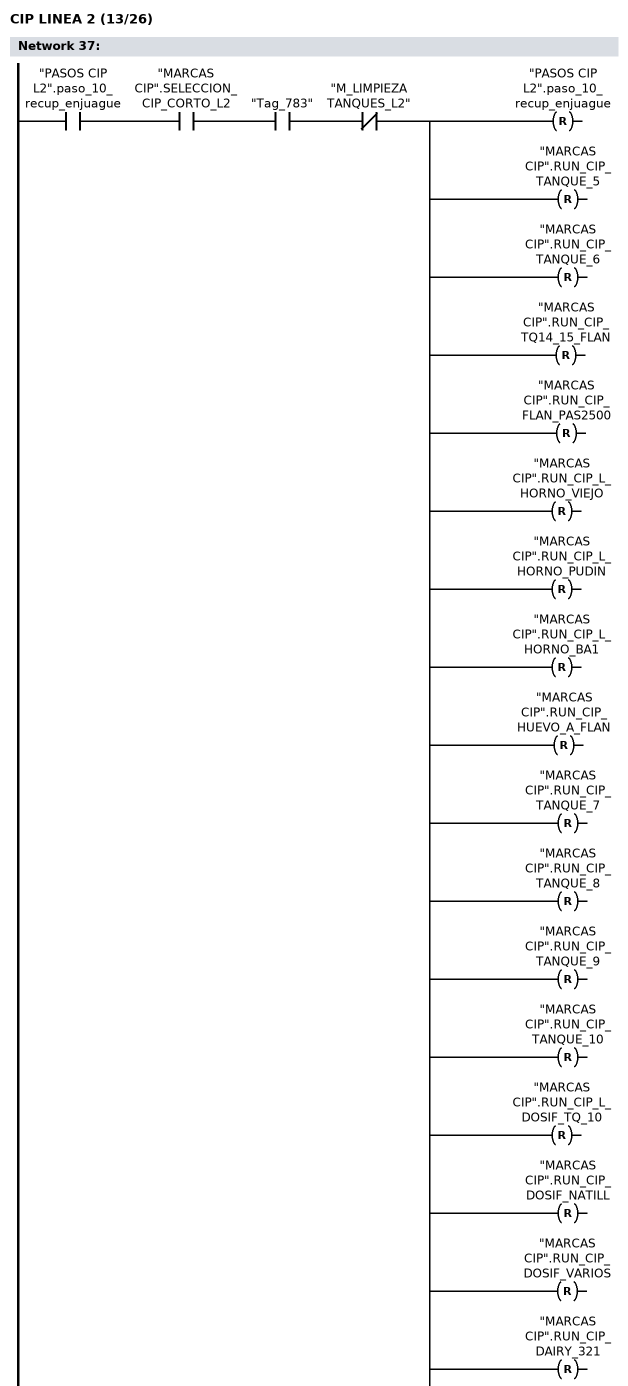
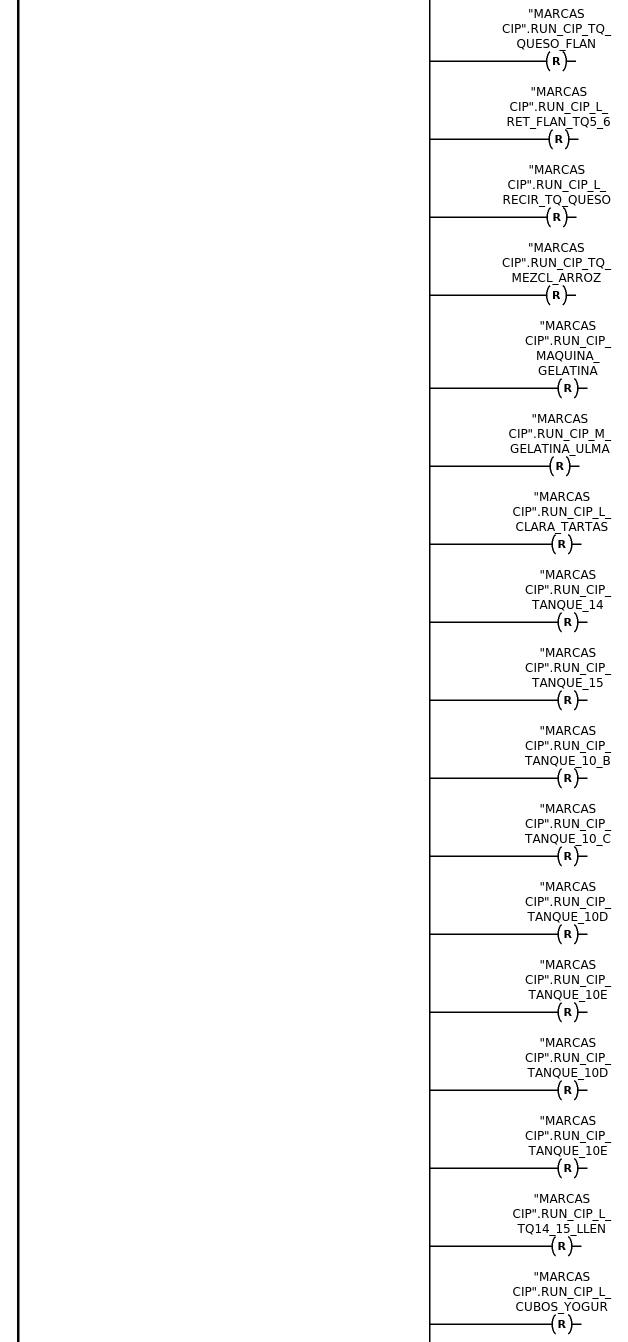
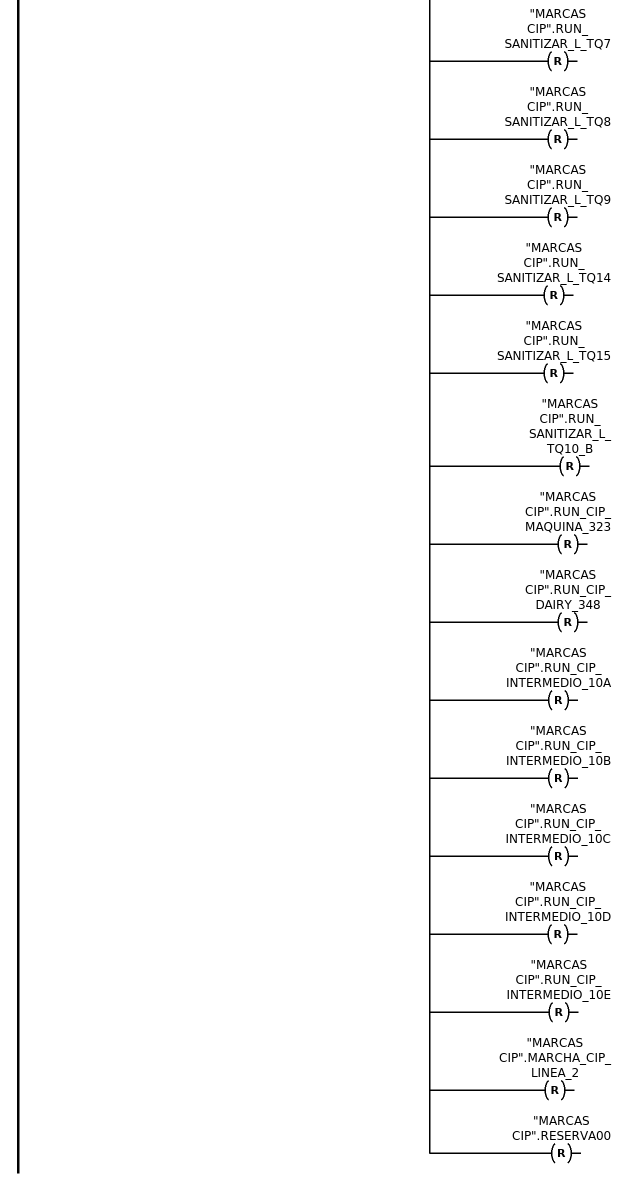
   RUNG wire#powerrail
      Contact( "PASOS CIP L2".paso_10_recup_enjuague )
      Contact( "MARCAS CIP".SELECCION_CIP_CORTO_L2 )
      Contact( "Tag_783" )
      I_Contact( "M_LIMPIEZA TANQUES_L2" )
      wire#w1
      R_Coil( "PASOS CIP L2".paso_10_recup_enjuague )
   END_RUNG
   RUNG wire#w1
      R_Coil( "MARCAS CIP".RUN_CIP_TANQUE_5 )
   END_RUNG
   RUNG wire#w1
      R_Coil( "MARCAS CIP".RUN_CIP_TANQUE_6 )
   END_RUNG
   RUNG wire#w1
      R_Coil( "MARCAS CIP".RUN_CIP_TQ14_15_FLAN )
   END_RUNG
   RUNG wire#w1
      R_Coil( "MARCAS CIP".RUN_CIP_FLAN_PAS2500 )
   END_RUNG
   RUNG wire#w1
      R_Coil( "MARCAS CIP".RUN_CIP_L_HORNO_VIEJO )
   END_RUNG
   RUNG wire#w1
      R_Coil( "MARCAS CIP".RUN_CIP_L_HORNO_PUDIN )
   END_RUNG
   RUNG wire#w1
      R_Coil( "MARCAS CIP".RUN_CIP_L_HORNO_BA1 )
   END_RUNG
   RUNG wire#w1
      R_Coil( "MARCAS CIP".RUN_CIP_HUEVO_A_FLAN )
   END_RUNG
   RUNG wire#w1
      R_Coil( "MARCAS CIP".RUN_CIP_TANQUE_7 )
   END_RUNG
   RUNG wire#w1
      R_Coil( "MARCAS CIP".RUN_CIP_TANQUE_8 )
   END_RUNG
   RUNG wire#w1
      R_Coil( "MARCAS CIP".RUN_CIP_TANQUE_9 )
   END_RUNG
   RUNG wire#w1
      R_Coil( "MARCAS CIP".RUN_CIP_TANQUE_10 )
   END_RUNG
   RUNG wire#w1
      R_Coil( "MARCAS CIP".RUN_CIP_L_DOSIF_TQ_10 )
   END_RUNG
   RUNG wire#w1
      R_Coil( "MARCAS CIP".RUN_CIP_DOSIF_NATILL )
   END_RUNG
   RUNG wire#w1
      R_Coil( "MARCAS CIP".RUN_CIP_DOSIF_VARIOS )
   END_RUNG
   RUNG wire#w1
      R_Coil( "MARCAS CIP".RUN_CIP_DAIRY_321 )
   END_RUNG
   RUNG wire#w1
      R_Coil( "MARCAS CIP".RUN_CIP_TQ_QUESO_FLAN )
   END_RUNG
   RUNG wire#w1
      R_Coil( "MARCAS CIP".RUN_CIP_L_RET_FLAN_TQ5_6 )
   END_RUNG
   RUNG wire#w1
      R_Coil( "MARCAS CIP".RUN_CIP_L_RECIR_TQ_QUESO )
   END_RUNG
   RUNG wire#w1
      R_Coil( "MARCAS CIP".RUN_CIP_TQ_MEZCL_ARROZ )
   END_RUNG
   RUNG wire#w1
      R_Coil( "MARCAS CIP".RUN_CIP_MAQUINA_GELATINA )
   END_RUNG
   RUNG wire#w1
      R_Coil( "MARCAS CIP".RUN_CIP_M_GELATINA_ULMA )
   END_RUNG
   RUNG wire#w1
      R_Coil( "MARCAS CIP".RUN_CIP_L_CLARA_TARTAS )
   END_RUNG
   RUNG wire#w1
      R_Coil( "MARCAS CIP".RUN_CIP_TANQUE_14 )
   END_RUNG
   RUNG wire#w1
      R_Coil( "MARCAS CIP".RUN_CIP_TANQUE_15 )
   END_RUNG
   RUNG wire#w1
      R_Coil( "MARCAS CIP".RUN_CIP_TANQUE_10_B )
   END_RUNG
   RUNG wire#w1
      R_Coil( "MARCAS CIP".RUN_CIP_TANQUE_10_C )
   END_RUNG
   RUNG wire#w1
      R_Coil( "MARCAS CIP".RUN_CIP_TANQUE_10D )
   END_RUNG
   RUNG wire#w1
      R_Coil( "MARCAS CIP".RUN_CIP_TANQUE_10E )
   END_RUNG
   RUNG wire#w1
      R_Coil( "MARCAS CIP".RUN_CIP_TANQUE_10D )
   END_RUNG
   RUNG wire#w1
      R_Coil( "MARCAS CIP".RUN_CIP_TANQUE_10E )
   END_RUNG
   RUNG wire#w1
      R_Coil( "MARCAS CIP".RUN_CIP_L_TQ14_15_LLEN )
   END_RUNG
   RUNG wire#w1
      R_Coil( "MARCAS CIP".RUN_CIP_L_CUBOS_YOGUR )
   END_RUNG
   RUNG wire#w1
      R_Coil( "MARCAS CIP".RUN_SANITIZAR_L_TQ7 )
   END_RUNG
   RUNG wire#w1
      R_Coil( "MARCAS CIP".RUN_SANITIZAR_L_TQ8 )
   END_RUNG
   RUNG wire#w1
      R_Coil( "MARCAS CIP".RUN_SANITIZAR_L_TQ9 )
   END_RUNG
   RUNG wire#w1
      R_Coil( "MARCAS CIP".RUN_SANITIZAR_L_TQ14 )
   END_RUNG
   RUNG wire#w1
      R_Coil( "MARCAS CIP".RUN_SANITIZAR_L_TQ15 )
   END_RUNG
   RUNG wire#w1
      R_Coil( "MARCAS CIP".RUN_SANITIZAR_L_TQ10_B )
   END_RUNG
   RUNG wire#w1
      R_Coil( "MARCAS CIP".RUN_CIP_MAQUINA_323 )
   END_RUNG
   RUNG wire#w1
      R_Coil( "MARCAS CIP".RUN_CIP_DAIRY_348 )
   END_RUNG
   RUNG wire#w1
      R_Coil( "MARCAS CIP".RUN_CIP_INTERMEDIO_10A )
   END_RUNG
   RUNG wire#w1
      R_Coil( "MARCAS CIP".RUN_CIP_INTERMEDIO_10B )
   END_RUNG
   RUNG wire#w1
      R_Coil( "MARCAS CIP".RUN_CIP_INTERMEDIO_10C )
   END_RUNG
   RUNG wire#w1
      R_Coil( "MARCAS CIP".RUN_CIP_INTERMEDIO_10D )
   END_RUNG
   RUNG wire#w1
      R_Coil( "MARCAS CIP".RUN_CIP_INTERMEDIO_10E )
   END_RUNG
   RUNG wire#w1
      R_Coil( "MARCAS CIP".MARCHA_CIP_LINEA_2 )
   END_RUNG
   RUNG wire#w1
      R_Coil( "MARCAS CIP".RESERVA00 )
   END_RUNG
   // the same network as SCL:
   #_w1 := "PASOS CIP L2".paso_10_recup_enjuague AND "MARCAS CIP".SELECCION_CIP_CORTO_L2 AND "Tag_783" AND NOT "M_LIMPIEZA TANQUES_L2";
   IF #_w1 THEN
       "PASOS CIP L2".paso_10_recup_enjuague := FALSE;
       "MARCAS CIP".RUN_CIP_TANQUE_5 := FALSE;
       "MARCAS CIP".RUN_CIP_TANQUE_6 := FALSE;
       "MARCAS CIP".RUN_CIP_TQ14_15_FLAN := FALSE;
       "MARCAS CIP".RUN_CIP_FLAN_PAS2500 := FALSE;
       "MARCAS CIP".RUN_CIP_L_HORNO_VIEJO := FALSE;
       "MARCAS CIP".RUN_CIP_L_HORNO_PUDIN := FALSE;
       "MARCAS CIP".RUN_CIP_L_HORNO_BA1 := FALSE;
       "MARCAS CIP".RUN_CIP_HUEVO_A_FLAN := FALSE;
       "MARCAS CIP".RUN_CIP_TANQUE_7 := FALSE;
       "MARCAS CIP".RUN_CIP_TANQUE_8 := FALSE;
       "MARCAS CIP".RUN_CIP_TANQUE_9 := FALSE;
       "MARCAS CIP".RUN_CIP_TANQUE_10 := FALSE;
       "MARCAS CIP".RUN_CIP_L_DOSIF_TQ_10 := FALSE;
       "MARCAS CIP".RUN_CIP_DOSIF_NATILL := FALSE;
       "MARCAS CIP".RUN_CIP_DOSIF_VARIOS := FALSE;
       "MARCAS CIP".RUN_CIP_DAIRY_321 := FALSE;
       "MARCAS CIP".RUN_CIP_TQ_QUESO_FLAN := FALSE;
       "MARCAS CIP".RUN_CIP_L_RET_FLAN_TQ5_6 := FALSE;
       "MARCAS CIP".RUN_CIP_L_RECIR_TQ_QUESO := FALSE;
       "MARCAS CIP".RUN_CIP_TQ_MEZCL_ARROZ := FALSE;
       "MARCAS CIP".RUN_CIP_MAQUINA_GELATINA := FALSE;
       "MARCAS CIP".RUN_CIP_M_GELATINA_ULMA := FALSE;
       "MARCAS CIP".RUN_CIP_L_CLARA_TARTAS := FALSE;
       "MARCAS CIP".RUN_CIP_TANQUE_14 := FALSE;
       "MARCAS CIP".RUN_CIP_TANQUE_15 := FALSE;
       "MARCAS CIP".RUN_CIP_TANQUE_10_B := FALSE;
       "MARCAS CIP".RUN_CIP_TANQUE_10_C := FALSE;
       "MARCAS CIP".RUN_CIP_TANQUE_10D := FALSE;
       "MARCAS CIP".RUN_CIP_TANQUE_10E := FALSE;
       "MARCAS CIP".RUN_CIP_TANQUE_10D := FALSE;
       "MARCAS CIP".RUN_CIP_TANQUE_10E := FALSE;
       "MARCAS CIP".RUN_CIP_L_TQ14_15_LLEN := FALSE;
       "MARCAS CIP".RUN_CIP_L_CUBOS_YOGUR := FALSE;
       "MARCAS CIP".RUN_SANITIZAR_L_TQ7 := FALSE;
       "MARCAS CIP".RUN_SANITIZAR_L_TQ8 := FALSE;
       "MARCAS CIP".RUN_SANITIZAR_L_TQ9 := FALSE;
       "MARCAS CIP".RUN_SANITIZAR_L_TQ14 := FALSE;
       "MARCAS CIP".RUN_SANITIZAR_L_TQ15 := FALSE;
       "MARCAS CIP".RUN_SANITIZAR_L_TQ10_B := FALSE;
       "MARCAS CIP".RUN_CIP_MAQUINA_323 := FALSE;
       "MARCAS CIP".RUN_CIP_DAIRY_348 := FALSE;
       "MARCAS CIP".RUN_CIP_INTERMEDIO_10A := FALSE;
       "MARCAS CIP".RUN_CIP_INTERMEDIO_10B := FALSE;
       "MARCAS CIP".RUN_CIP_INTERMEDIO_10C := FALSE;
       "MARCAS CIP".RUN_CIP_INTERMEDIO_10D := FALSE;
       "MARCAS CIP".RUN_CIP_INTERMEDIO_10E := FALSE;
       "MARCAS CIP".MARCHA_CIP_LINEA_2 := FALSE;
       "MARCAS CIP".RESERVA00 := FALSE;
   END_IF;
END_REGION

REGION Network 38: PASO 11: VACIADO SI TANQUE
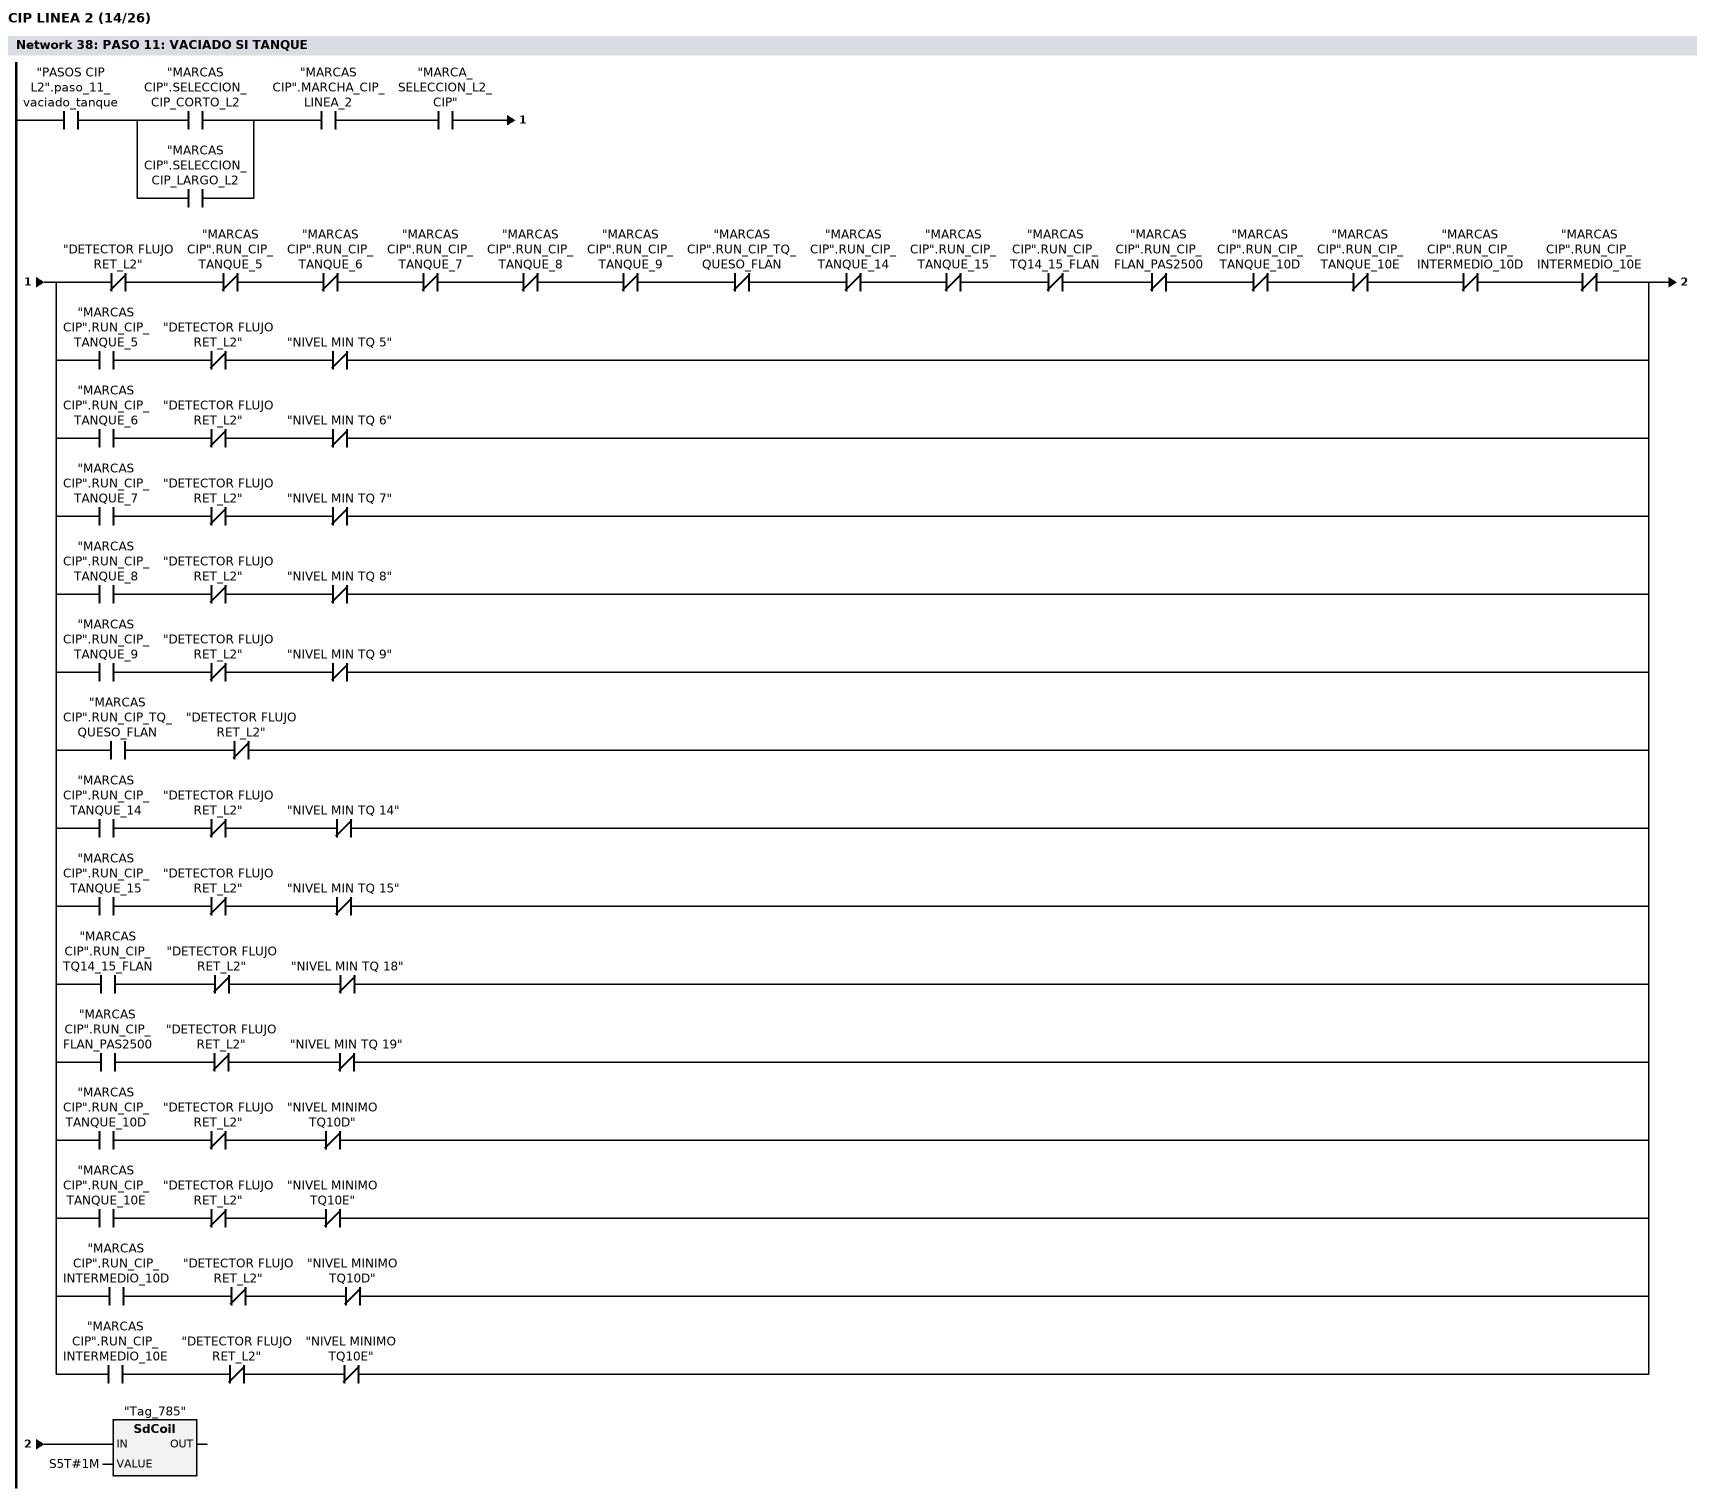
   // no SCL statement known for SdCoil: written as a call
   SdCoil(value := S5T#1M,
          in := "PASOS CIP L2".paso_11_vaciado_tanque AND ("MARCAS CIP".SELECCION_CIP_CORTO_L2 OR "MARCAS CIP".SELECCION_CIP_LARGO_L2) AND "MARCAS CIP".MARCHA_CIP_LINEA_2 AND "MARCA_SELECCION_L2_CIP" AND ((NOT "DETECTOR FLUJO RET_L2" AND NOT "MARCAS CIP".RUN_CIP_TANQUE_5 AND NOT "MARCAS CIP".RUN_CIP_TANQUE_6 AND NOT "MARCAS CIP".RUN_CIP_TANQUE_7 AND NOT "MARCAS CIP".RUN_CIP_TANQUE_8 AND NOT "MARCAS CIP".RUN_CIP_TANQUE_9 AND NOT "MARCAS CIP".RUN_CIP_TQ_QUESO_FLAN AND NOT "MARCAS CIP".RUN_CIP_TANQUE_14 AND NOT "MARCAS CIP".RUN_CIP_TANQUE_15 AND NOT "MARCAS CIP".RUN_CIP_TQ14_15_FLAN AND NOT "MARCAS CIP".RUN_CIP_FLAN_PAS2500 AND NOT "MARCAS CIP".RUN_CIP_TANQUE_10D AND NOT "MARCAS CIP".RUN_CIP_TANQUE_10E AND NOT "MARCAS CIP".RUN_CIP_INTERMEDIO_10D AND NOT "MARCAS CIP".RUN_CIP_INTERMEDIO_10E) OR ("MARCAS CIP".RUN_CIP_TANQUE_5 AND NOT "DETECTOR FLUJO RET_L2" AND NOT "NIVEL MIN TQ 5") OR ("MARCAS CIP".RUN_CIP_TANQUE_6 AND NOT "DETECTOR FLUJO RET_L2" AND NOT "NIVEL MIN TQ 6") OR ("MARCAS CIP".RUN_CIP_TANQUE_7 AND NOT "DETECTOR FLUJO RET_L2" AND NOT "NIVEL MIN TQ 7") OR ("MARCAS CIP".RUN_CIP_TANQUE_8 AND NOT "DETECTOR FLUJO RET_L2" AND NOT "NIVEL MIN TQ 8") OR ("MARCAS CIP".RUN_CIP_TANQUE_9 AND NOT "DETECTOR FLUJO RET_L2" AND NOT "NIVEL MIN TQ 9") OR ("MARCAS CIP".RUN_CIP_TQ_QUESO_FLAN AND NOT "DETECTOR FLUJO RET_L2") OR ("MARCAS CIP".RUN_CIP_TANQUE_14 AND NOT "DETECTOR FLUJO RET_L2" AND NOT "NIVEL MIN TQ 14") OR ("MARCAS CIP".RUN_CIP_TANQUE_15 AND NOT "DETECTOR FLUJO RET_L2" AND NOT "NIVEL MIN TQ 15") OR ("MARCAS CIP".RUN_CIP_TQ14_15_FLAN AND NOT "DETECTOR FLUJO RET_L2" AND NOT "NIVEL MIN TQ 18") OR ("MARCAS CIP".RUN_CIP_FLAN_PAS2500 AND NOT "DETECTOR FLUJO RET_L2" AND NOT "NIVEL MIN TQ 19") OR ("MARCAS CIP".RUN_CIP_TANQUE_10D AND NOT "DETECTOR FLUJO RET_L2" AND NOT "NIVEL MINIMO TQ10D") OR ("MARCAS CIP".RUN_CIP_TANQUE_10E AND NOT "DETECTOR FLUJO RET_L2" AND NOT "NIVEL MINIMO TQ10E") OR ("MARCAS CIP".RUN_CIP_INTERMEDIO_10D AND NOT "DETECTOR FLUJO RET_L2" AND NOT "NIVEL MINIMO TQ10D") OR ("MARCAS CIP".RUN_CIP_INTERMEDIO_10E AND NOT "DETECTOR FLUJO RET_L2" AND NOT "NIVEL MINIMO TQ10E")),
          operand := "Tag_785");
END_REGION

REGION Network 39
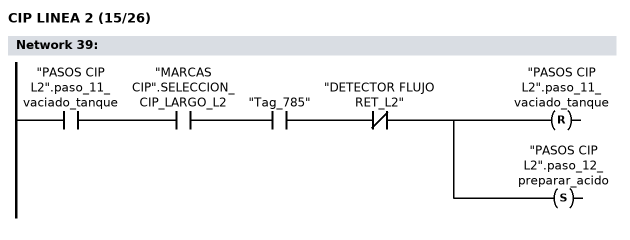
   RUNG wire#powerrail
      Contact( "PASOS CIP L2".paso_11_vaciado_tanque )
      Contact( "MARCAS CIP".SELECCION_CIP_LARGO_L2 )
      Contact( "Tag_785" )
      I_Contact( "DETECTOR FLUJO RET_L2" )
      wire#w1
      R_Coil( "PASOS CIP L2".paso_11_vaciado_tanque )
   END_RUNG
   RUNG wire#w1
      S_Coil( "PASOS CIP L2".paso_12_preparar_acido )
   END_RUNG
   // the same network as SCL:
   #_w1 := "PASOS CIP L2".paso_11_vaciado_tanque AND "MARCAS CIP".SELECCION_CIP_LARGO_L2 AND "Tag_785" AND NOT "DETECTOR FLUJO RET_L2";
   IF #_w1 THEN
       "PASOS CIP L2".paso_11_vaciado_tanque := FALSE;
       "PASOS CIP L2".paso_12_preparar_acido := TRUE;
   END_IF;
END_REGION

REGION Network 40
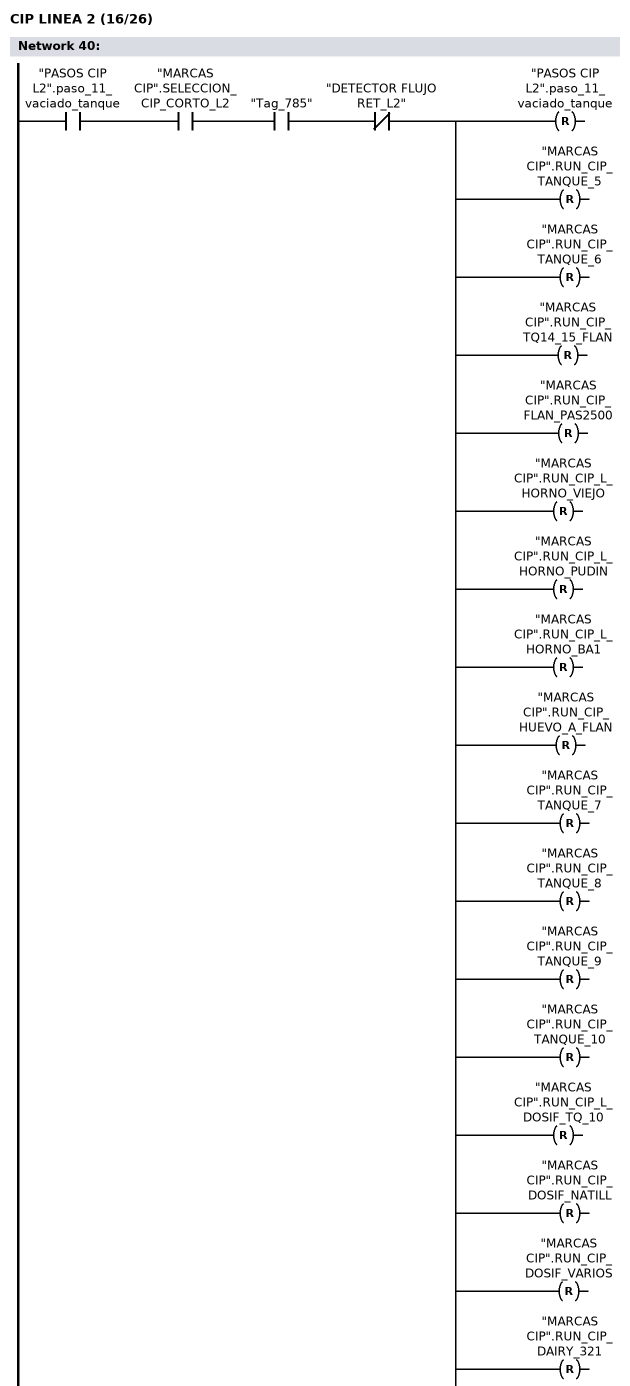
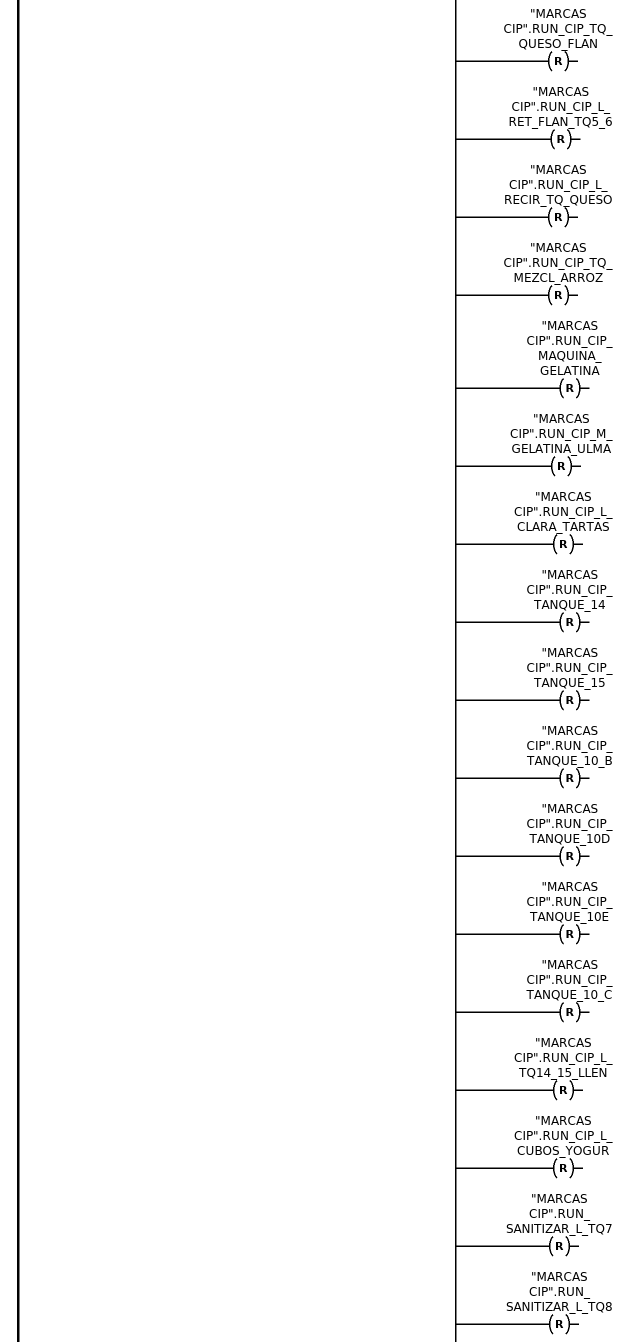
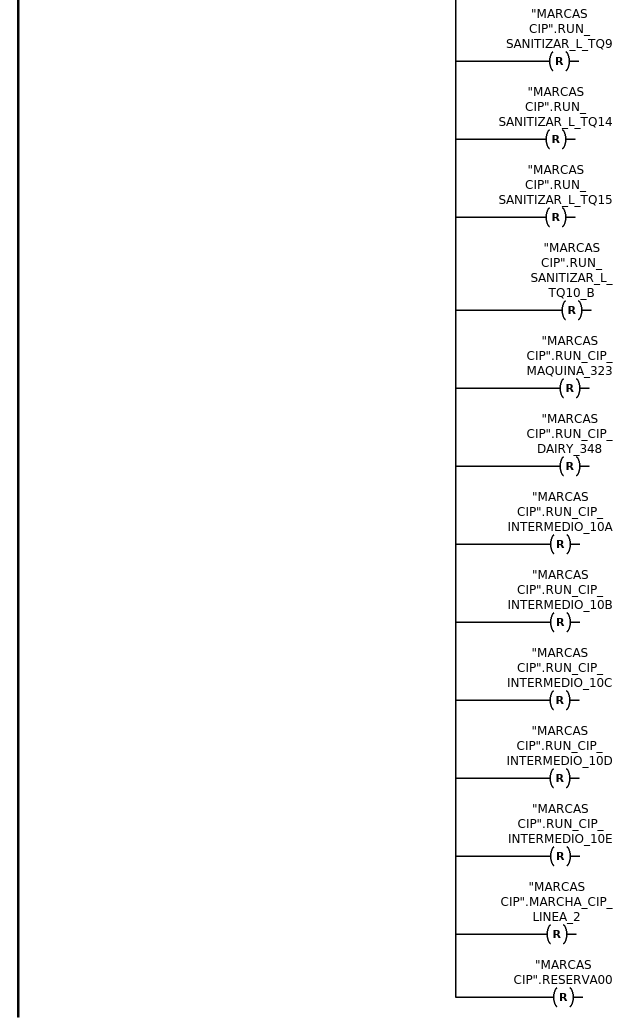
   RUNG wire#powerrail
      Contact( "PASOS CIP L2".paso_11_vaciado_tanque )
      Contact( "MARCAS CIP".SELECCION_CIP_CORTO_L2 )
      Contact( "Tag_785" )
      I_Contact( "DETECTOR FLUJO RET_L2" )
      wire#w1
      R_Coil( "PASOS CIP L2".paso_11_vaciado_tanque )
   END_RUNG
   RUNG wire#w1
      R_Coil( "MARCAS CIP".RUN_CIP_TANQUE_5 )
   END_RUNG
   RUNG wire#w1
      R_Coil( "MARCAS CIP".RUN_CIP_TANQUE_6 )
   END_RUNG
   RUNG wire#w1
      R_Coil( "MARCAS CIP".RUN_CIP_TQ14_15_FLAN )
   END_RUNG
   RUNG wire#w1
      R_Coil( "MARCAS CIP".RUN_CIP_FLAN_PAS2500 )
   END_RUNG
   RUNG wire#w1
      R_Coil( "MARCAS CIP".RUN_CIP_L_HORNO_VIEJO )
   END_RUNG
   RUNG wire#w1
      R_Coil( "MARCAS CIP".RUN_CIP_L_HORNO_PUDIN )
   END_RUNG
   RUNG wire#w1
      R_Coil( "MARCAS CIP".RUN_CIP_L_HORNO_BA1 )
   END_RUNG
   RUNG wire#w1
      R_Coil( "MARCAS CIP".RUN_CIP_HUEVO_A_FLAN )
   END_RUNG
   RUNG wire#w1
      R_Coil( "MARCAS CIP".RUN_CIP_TANQUE_7 )
   END_RUNG
   RUNG wire#w1
      R_Coil( "MARCAS CIP".RUN_CIP_TANQUE_8 )
   END_RUNG
   RUNG wire#w1
      R_Coil( "MARCAS CIP".RUN_CIP_TANQUE_9 )
   END_RUNG
   RUNG wire#w1
      R_Coil( "MARCAS CIP".RUN_CIP_TANQUE_10 )
   END_RUNG
   RUNG wire#w1
      R_Coil( "MARCAS CIP".RUN_CIP_L_DOSIF_TQ_10 )
   END_RUNG
   RUNG wire#w1
      R_Coil( "MARCAS CIP".RUN_CIP_DOSIF_NATILL )
   END_RUNG
   RUNG wire#w1
      R_Coil( "MARCAS CIP".RUN_CIP_DOSIF_VARIOS )
   END_RUNG
   RUNG wire#w1
      R_Coil( "MARCAS CIP".RUN_CIP_DAIRY_321 )
   END_RUNG
   RUNG wire#w1
      R_Coil( "MARCAS CIP".RUN_CIP_TQ_QUESO_FLAN )
   END_RUNG
   RUNG wire#w1
      R_Coil( "MARCAS CIP".RUN_CIP_L_RET_FLAN_TQ5_6 )
   END_RUNG
   RUNG wire#w1
      R_Coil( "MARCAS CIP".RUN_CIP_L_RECIR_TQ_QUESO )
   END_RUNG
   RUNG wire#w1
      R_Coil( "MARCAS CIP".RUN_CIP_TQ_MEZCL_ARROZ )
   END_RUNG
   RUNG wire#w1
      R_Coil( "MARCAS CIP".RUN_CIP_MAQUINA_GELATINA )
   END_RUNG
   RUNG wire#w1
      R_Coil( "MARCAS CIP".RUN_CIP_M_GELATINA_ULMA )
   END_RUNG
   RUNG wire#w1
      R_Coil( "MARCAS CIP".RUN_CIP_L_CLARA_TARTAS )
   END_RUNG
   RUNG wire#w1
      R_Coil( "MARCAS CIP".RUN_CIP_TANQUE_14 )
   END_RUNG
   RUNG wire#w1
      R_Coil( "MARCAS CIP".RUN_CIP_TANQUE_15 )
   END_RUNG
   RUNG wire#w1
      R_Coil( "MARCAS CIP".RUN_CIP_TANQUE_10_B )
   END_RUNG
   RUNG wire#w1
      R_Coil( "MARCAS CIP".RUN_CIP_TANQUE_10D )
   END_RUNG
   RUNG wire#w1
      R_Coil( "MARCAS CIP".RUN_CIP_TANQUE_10E )
   END_RUNG
   RUNG wire#w1
      R_Coil( "MARCAS CIP".RUN_CIP_TANQUE_10_C )
   END_RUNG
   RUNG wire#w1
      R_Coil( "MARCAS CIP".RUN_CIP_L_TQ14_15_LLEN )
   END_RUNG
   RUNG wire#w1
      R_Coil( "MARCAS CIP".RUN_CIP_L_CUBOS_YOGUR )
   END_RUNG
   RUNG wire#w1
      R_Coil( "MARCAS CIP".RUN_SANITIZAR_L_TQ7 )
   END_RUNG
   RUNG wire#w1
      R_Coil( "MARCAS CIP".RUN_SANITIZAR_L_TQ8 )
   END_RUNG
   RUNG wire#w1
      R_Coil( "MARCAS CIP".RUN_SANITIZAR_L_TQ9 )
   END_RUNG
   RUNG wire#w1
      R_Coil( "MARCAS CIP".RUN_SANITIZAR_L_TQ14 )
   END_RUNG
   RUNG wire#w1
      R_Coil( "MARCAS CIP".RUN_SANITIZAR_L_TQ15 )
   END_RUNG
   RUNG wire#w1
      R_Coil( "MARCAS CIP".RUN_SANITIZAR_L_TQ10_B )
   END_RUNG
   RUNG wire#w1
      R_Coil( "MARCAS CIP".RUN_CIP_MAQUINA_323 )
   END_RUNG
   RUNG wire#w1
      R_Coil( "MARCAS CIP".RUN_CIP_DAIRY_348 )
   END_RUNG
   RUNG wire#w1
      R_Coil( "MARCAS CIP".RUN_CIP_INTERMEDIO_10A )
   END_RUNG
   RUNG wire#w1
      R_Coil( "MARCAS CIP".RUN_CIP_INTERMEDIO_10B )
   END_RUNG
   RUNG wire#w1
      R_Coil( "MARCAS CIP".RUN_CIP_INTERMEDIO_10C )
   END_RUNG
   RUNG wire#w1
      R_Coil( "MARCAS CIP".RUN_CIP_INTERMEDIO_10D )
   END_RUNG
   RUNG wire#w1
      R_Coil( "MARCAS CIP".RUN_CIP_INTERMEDIO_10E )
   END_RUNG
   RUNG wire#w1
      R_Coil( "MARCAS CIP".MARCHA_CIP_LINEA_2 )
   END_RUNG
   RUNG wire#w1
      R_Coil( "MARCAS CIP".RESERVA00 )
   END_RUNG
   // the same network as SCL:
   #_w1 := "PASOS CIP L2".paso_11_vaciado_tanque AND "MARCAS CIP".SELECCION_CIP_CORTO_L2 AND "Tag_785" AND NOT "DETECTOR FLUJO RET_L2";
   IF #_w1 THEN
       "PASOS CIP L2".paso_11_vaciado_tanque := FALSE;
       "MARCAS CIP".RUN_CIP_TANQUE_5 := FALSE;
       "MARCAS CIP".RUN_CIP_TANQUE_6 := FALSE;
       "MARCAS CIP".RUN_CIP_TQ14_15_FLAN := FALSE;
       "MARCAS CIP".RUN_CIP_FLAN_PAS2500 := FALSE;
       "MARCAS CIP".RUN_CIP_L_HORNO_VIEJO := FALSE;
       "MARCAS CIP".RUN_CIP_L_HORNO_PUDIN := FALSE;
       "MARCAS CIP".RUN_CIP_L_HORNO_BA1 := FALSE;
       "MARCAS CIP".RUN_CIP_HUEVO_A_FLAN := FALSE;
       "MARCAS CIP".RUN_CIP_TANQUE_7 := FALSE;
       "MARCAS CIP".RUN_CIP_TANQUE_8 := FALSE;
       "MARCAS CIP".RUN_CIP_TANQUE_9 := FALSE;
       "MARCAS CIP".RUN_CIP_TANQUE_10 := FALSE;
       "MARCAS CIP".RUN_CIP_L_DOSIF_TQ_10 := FALSE;
       "MARCAS CIP".RUN_CIP_DOSIF_NATILL := FALSE;
       "MARCAS CIP".RUN_CIP_DOSIF_VARIOS := FALSE;
       "MARCAS CIP".RUN_CIP_DAIRY_321 := FALSE;
       "MARCAS CIP".RUN_CIP_TQ_QUESO_FLAN := FALSE;
       "MARCAS CIP".RUN_CIP_L_RET_FLAN_TQ5_6 := FALSE;
       "MARCAS CIP".RUN_CIP_L_RECIR_TQ_QUESO := FALSE;
       "MARCAS CIP".RUN_CIP_TQ_MEZCL_ARROZ := FALSE;
       "MARCAS CIP".RUN_CIP_MAQUINA_GELATINA := FALSE;
       "MARCAS CIP".RUN_CIP_M_GELATINA_ULMA := FALSE;
       "MARCAS CIP".RUN_CIP_L_CLARA_TARTAS := FALSE;
       "MARCAS CIP".RUN_CIP_TANQUE_14 := FALSE;
       "MARCAS CIP".RUN_CIP_TANQUE_15 := FALSE;
       "MARCAS CIP".RUN_CIP_TANQUE_10_B := FALSE;
       "MARCAS CIP".RUN_CIP_TANQUE_10D := FALSE;
       "MARCAS CIP".RUN_CIP_TANQUE_10E := FALSE;
       "MARCAS CIP".RUN_CIP_TANQUE_10_C := FALSE;
       "MARCAS CIP".RUN_CIP_L_TQ14_15_LLEN := FALSE;
       "MARCAS CIP".RUN_CIP_L_CUBOS_YOGUR := FALSE;
       "MARCAS CIP".RUN_SANITIZAR_L_TQ7 := FALSE;
       "MARCAS CIP".RUN_SANITIZAR_L_TQ8 := FALSE;
       "MARCAS CIP".RUN_SANITIZAR_L_TQ9 := FALSE;
       "MARCAS CIP".RUN_SANITIZAR_L_TQ14 := FALSE;
       "MARCAS CIP".RUN_SANITIZAR_L_TQ15 := FALSE;
       "MARCAS CIP".RUN_SANITIZAR_L_TQ10_B := FALSE;
       "MARCAS CIP".RUN_CIP_MAQUINA_323 := FALSE;
       "MARCAS CIP".RUN_CIP_DAIRY_348 := FALSE;
       "MARCAS CIP".RUN_CIP_INTERMEDIO_10A := FALSE;
       "MARCAS CIP".RUN_CIP_INTERMEDIO_10B := FALSE;
       "MARCAS CIP".RUN_CIP_INTERMEDIO_10C := FALSE;
       "MARCAS CIP".RUN_CIP_INTERMEDIO_10D := FALSE;
       "MARCAS CIP".RUN_CIP_INTERMEDIO_10E := FALSE;
       "MARCAS CIP".MARCHA_CIP_LINEA_2 := FALSE;
       "MARCAS CIP".RESERVA00 := FALSE;
   END_IF;
END_REGION

REGION Network 41
